METHOD FB_init : BOOL
VAR_INPUT
	bInitRetains : BOOL; // if TRUE, the retain variables are initialized (warm start / cold start)
	bInCopyCode : BOOL;  // if TRUE, the instance afterwards gets moved into the copy code (online change)
END_VAR
nHighestPumpNr := nHighestPumpNr + 1;
nPumpNr := nHighestPumpNr;
END_METHOD

ACTION A_PumpConst:
//Egal in welchem State, wenn Flow neu gesetzt wird, dann Rotate neu senden
//Wenn bStop, in jedem State zu Stop gehen

IF nStateA_Pump = 0 THEN
	nPumpSpeed := nPumpSpeedNew;
	nStateA_Pump := 1;
END_IF

CASE nStateA_Pump OF
	1:	//Motor rechts drehen
		fbTMCM6110(bExecute:= TRUE, eCommand:= E_TMCMCommand.ROTATE_R, nSendValue:= nPumpSpeed, nMotorNr:= nPumpNr);
		IF NOT fbTMCM6110.bBusy THEN
			IF fbTMCM6110.bError THEN
				nStateA_Pump := 99;	
			ELSE
				IF nPumpSpeed = nPumpSpeedNew THEN
					nStateA_Pump := 2;
				ELSE
					nStateA_Pump := 0;
				END_IF
			END_IF
			fbTMCM6110(bExecute:= FALSE, nMotorNr:= nPumpNr);
		END_IF
		
	2:	//IstSpeed abfragen
		fbTMCM6110(bExecute:= TRUE, eCommand:= E_TMCMCommand.GET_ACT_SPEED, nMotorNr:= nPumpNr);
		IF NOT fbTMCM6110.bBusy THEN
			IF fbTMCM6110.bError THEN
				nStateA_Pump := 99;	
			ELSE
				IF nPumpSpeed <> nPumpSpeedNew THEN
					nStateA_Pump := 0;
				ELSE
					IF fbTMCM6110.nReceiveValue = nPumpSpeed THEN	//SollSpeed erreicht
						IF nPumpSpeed = 0 THEN
							nStateA_Pump := 80;
						END_IF
					END_IF
				END_IF
			END_IF
			fbTMCM6110(bExecute:= FALSE, nMotorNr:= nPumpNr);
		END_IF
END_CASE
END_ACTION

METHOD M_Stop : ERRORID
VAR_INPUT
END_VAR
IF bBusy THEN
	bStop := TRUE;
	nPumpSpeedNew := 0;
END_IF
END_METHOD

ACTION A_PumpQuantity:
//Wenn bStop, in jedem State zu Stop gehen
//Vor Absenden des Move-Befehls, Speed setzen
CASE nStateA_Pump OF
	
	0:	//Set Speed
		nPumpSpeed := nPumpSpeedNew;
		fbTMCM6110(bExecute:= TRUE, eCommand:= E_TMCMCommand.SET_SPEED, nSendValue:= nPumpSpeed, nMotorNr:= nPumpNr);
		IF NOT fbTMCM6110.bBusy THEN
			IF fbTMCM6110.bError THEN
				nStateA_Pump := 99;	
			ELSE
				IF bStop THEN
					nStateA_Pump := 80;
				ELSE
					nStateA_Pump := 1;
				END_IF
			END_IF
			fbTMCM6110(bExecute:= FALSE, nMotorNr:= nPumpNr);
		END_IF
		
	1:	//MoveRel
		fbTMCM6110(bExecute:= TRUE, eCommand:= E_TMCMCommand.MOVE_REL, nSendValue:= nPumpMicroSteps, nMotorNr:= nPumpNr);
		IF NOT fbTMCM6110.bBusy THEN
			IF fbTMCM6110.bError THEN
				nStateA_Pump := 99;	
			ELSE
				IF bStop THEN
					nStateA_Pump := 3;
				ELSE
					nStateA_Pump := 2;
				END_IF
			END_IF
			fbTMCM6110(bExecute:= FALSE, nMotorNr:= nPumpNr);
		END_IF
		
	2:	//Warten, bis Position erreicht
		fbTMCM6110(bExecute:= TRUE, eCommand:= E_TMCMCommand.GET_POS_REACHED, nSendValue:= 0, nMotorNr:= nPumpNr);
		IF NOT fbTMCM6110.bBusy THEN
			IF fbTMCM6110.bError THEN
				nStateA_Pump := 99;	
			ELSE
				IF bStop THEN
					nStateA_Pump := 3;	//Stoppen
				ELSE
					IF fbTMCM6110.nReceiveValue = 1 THEN
						nStateA_Pump := 80;	
					END_IF
				END_IF
			END_IF
			fbTMCM6110(bExecute:= FALSE, nMotorNr:= nPumpNr);
		END_IF
		
	3:	//Stoppen
		fbTMCM6110(bExecute:= TRUE, eCommand:= E_TMCMCommand.STOP, nSendValue:= 0, nMotorNr:= nPumpNr);
		IF NOT fbTMCM6110.bBusy THEN
			IF fbTMCM6110.bError THEN
				nStateA_Pump := 99;	
			ELSE
				nStateA_Pump := 80;	
			END_IF
			fbTMCM6110(bExecute:= FALSE, nMotorNr:= nPumpNr);
		END_IF
		
END_CASE
END_ACTION

METHOD M_PumpQuantity : ERRORID
VAR_INPUT
	nQuantity 	: DINT;
	nFlow		: DINT;
END_VAR
bPumpQuantity := TRUE;
nPumpMicroSteps := REAL_TO_DINT(DINT_TO_REAL(nQuantity) * cFactorQuantToMicroSteps);
nPumpSpeedNew := REAL_TO_DINT(DINT_TO_REAL(nFlow) * cFactorFlowToSpeed / cDivisorFlowToSpeed);
bBusy := TRUE;
END_METHOD

END_FUNCTION_BLOCK

// ---- Hardware/LiquidReserve/FB_TMCM6110.TcPOU
FUNCTION_BLOCK FB_TMCM6110
VAR_INPUT
	bExecute	: BOOL;
	eCommand	: E_TMCMCommand;
	nSendValue	: DINT;	
END_VAR
VAR_IN_OUT
	nMotorNr : USINT;
END_VAR
VAR_OUTPUT
	bBusy			: BOOL;
	bError			: BOOL;
	nReceiveValue	: DINT;	
END_VAR
VAR
	fbSendCanMessage 		: FB_SendCanMessage(ADR(CANInterfaceCom.stCanInterfaceBuffer));
	nState					: USINT;
	uByteArr4Dint			: U_ByteArr4_DINT;
END_VAR

IF bExecute THEN

	IF nState = 0 THEN
		bBusy := TRUE;
		fbSendCanMessage.aTxData[0] := UINT_TO_USINT(SHR(eCommand,8)); //Command
		fbSendCanMessage.aTxData[1] := UINT_TO_USINT(eCommand AND 16#00FF); //Type
		fbSendCanMessage.aTxData[2] := nMotorNr - 1; // "0" für Motor1
		//SendValue in Union kopieren
		uByteArr4Dint.nDINT := nSendValue;
		//Bytes aus Union in TxData kopieren (MSB in Byte3....LSB in Byte6)
		fbSendCanMessage.aTxData[3] := uByteArr4Dint.aBytes[3];
		fbSendCanMessage.aTxData[4] := uByteArr4Dint.aBytes[2];
		fbSendCanMessage.aTxData[5] := uByteArr4Dint.aBytes[1];
		fbSendCanMessage.aTxData[6] := uByteArr4Dint.aBytes[0];
		fbSendCanMessage.tTimeout := T#100MS;
		fbSendCanMessage.nTxLength := 8;
		nState := 60;
	END_IF
	
	IF nState = 60 THEN
		fbSendCanMessage(nIdentifierTX:= 16#01, nIdentifierRX:= 16#02, bExecute:= TRUE);
		IF NOT fbSendCanMessage.bBusy THEN
			IF NOT fbSendCanMessage.bError THEN
				//Response auswerten
				IF fbSendCanMessage.aRxData[1] = 100 THEN	//OK ohne Fehler
					//Bytes aus RxData in UNION kopieren (Byte3 in MSB....Byte6 in LSB)
					uByteArr4Dint.aBytes[3] := fbSendCanMessage.aRxData[3];
					uByteArr4Dint.aBytes[2] := fbSendCanMessage.aRxData[4];
					uByteArr4Dint.aBytes[1] := fbSendCanMessage.aRxData[5];
					uByteArr4Dint.aBytes[0] := fbSendCanMessage.aRxData[6];
					//nDint aus UNION in nReceiveValue koipieren
					nReceiveValue := uByteArr4Dint.nDINT;
					nState := 80;
				ELSE
					nState := 99;	
				END_IF
			ELSE
				nState := 99;
			END_IF
			fbSendCanMessage(bExecute:= FALSE);
		END_IF		
	END_IF
	
	IF nState = 80 THEN
		bBusy := FALSE;
	ELSIF nState = 99 THEN
		bBusy := FALSE;
		bError := TRUE;
	END_IF
	
ELSE
	bError := FALSE;
	nState := 0;
	nSendValue := 0;
	nReceiveValue := 0;
END_IF

END_FUNCTION_BLOCK

// ---- Hardware/FBox/FB_HwRefMultiPurpIO.TcPOU
FUNCTION_BLOCK FB_HwRefMultiPurpIO EXTENDS FB_CanNodeBase
VAR_INPUT
END_VAR
VAR_OUTPUT
END_VAR
VAR
END_VAR

IF bNodeEnabled THEN
	SUPER^();
END_IF

//Wenn die analogen Eingänge gemappt sind, dann müssen diese enabled werden.
//Hier sind diese allerdings nicht verfügbar. Wie komme ich an den Mapping-Status?
//IF F_GetMappingStatus(

ACTION A_ResetApp:
IF nStateA_ResetApp = 0 THEN
	fbSdoWrite(sADSNetID:= stAdsAdress.sNetId, nPortNr:= stAdsAdress.nPort,
				nIndex := cUpdateRequest.nIndex, nSubIndex := 0, nDataLength := 1, nData:= 1, bExecute:= TRUE);
	IF NOT fbSdoWrite.bBusy THEN
		IF fbSdoWrite.bError THEN
			nErrorId := fbSdoWrite.nAdsErrorId;
			nErrorId2 := fbSdoWrite.nSdoErrorId;
			nStateA_ResetApp := 99;  //Error
		ELSE
			nStateA_ResetApp := 80;
		END_IF
		fbSdoWrite(bExecute:= FALSE);
	END_IF
END_IF
END_ACTION

END_FUNCTION_BLOCK

// ---- Hardware/FBox/FB_PCV.TcPOU
FUNCTION_BLOCK FB_PCV
VAR_INPUT
END_VAR
VAR_OUTPUT
	bError : BOOL;
	nErrorId : ERRORID;
END_VAR
VAR
	bFill		: BOOL;
	tmrTimeout	: TON;
	bSensor		AT %I* : BOOL; 	//Verknüpfung mit Füllstandssensor
	bDigiOut 	AT %Q* : BOOL; 	//Verknüpfung muss mit Pumpe und StopVentil erfolgen
	bPneuValve	AT %Q* : BOOL;	//Verknüpfung mit Pneumatikventil (nur bei SolenoidPip)	
END_VAR

IF bSensor AND bFill THEN
	{IF defined(variable:cLiquidBottleNrPCV)}
	IF NOT aSensSysLiquidBottle[cLiquidBottleNrPCV] THEN //kein Systemwasser vorhanden
		bError := TRUE;
		nErrorId := E_ErrorIdCmd.ERRORID_LiquidBottleEmpty;
	END_IF
	{ELSE}
	IF NOT aSensSysLiquidBottle[1] THEN //kein Systemwasser vorhanden
		bError := TRUE;
		nErrorId := E_ErrorIdCmd.ERRORID_LiquidBottleEmpty;
	END_IF	
	{END_IF}

	IF NOT bError AND bFill THEN
		tmrTimeout(IN:= TRUE, PT:=T#1M);
		bDigiOut := TRUE;
	ELSE
		tmrTimeout(IN:= FALSE);
		bDigiOut := FALSE;	
	END_IF

	bFill := FALSE;
ELSE
	tmrTimeout(IN:= FALSE);
	bDigiOut := FALSE;	
	tmrTimeout(IN:= FALSE);
END_IF

IF tmrTimeout.Q THEN
	bError := TRUE;
	nErrorId := E_ErrorIdCmd.ERRORID_TimeOutFillPCV;
	bDigiOut := FALSE;
END_IF

METHOD M_Fill
VAR_INPUT
END_VAR
bFill := TRUE;
END_METHOD

METHOD M_Reset
VAR_INPUT
END_VAR
bError := FALSE;
END_METHOD

METHOD M_SwitchPneuValve
VAR_INPUT
	bOn : BOOL;
END_VAR
bPneuValve := bOn;
END_METHOD

PROPERTY P_bPneuValve : BOOL
GET
P_bPneuValve := bPneuValve;
END_GET
END_PROPERTY

END_FUNCTION_BLOCK

// ---- Hardware/Safety/FB_Safety.TcPOU
FUNCTION_BLOCK FB_Safety  EXTENDS FB_SafetyBase

VAR_INPUT
END_VAR

VAR_OUTPUT
	bVoltageSafe			: BOOL;
	bToolTempSafe			: BOOL;
END_VAR

VAR
	bEmergencyStop			AT %I* : BOOL;	//Notaus ist gedrückt
	bInterlockIsLocked		AT %I* : BOOL;	//Interlock ist ordnungsgemäß verriegelt
	bBoxContactsClosed		AT %I* : BOOL;	//Sicherheitskontakte der Sicherheitsbox geschlossen
	bDriveIsSafe			AT %I* : BOOL;	//Sicherheitsrelais der Antriebe haben nicht angezogen
	bMesIsSafe				AT %I* : BOOL;	//Sicherheitsrelais in MES-Box hat nicht angezogen
	 
	nTwinSafeGrpState		AT %I* : USINT;
	
	bRequDriveOn			AT %Q* : BOOL;	//Request an TwinSafe Gruppe die Drives freizugeben (Relais einschalten)
	bRequMesOn				AT %Q* : BOOL;	//Request an TwinSafe Gruppe die MES freizugeben (Relais im HV-Generator einschalten)
	bRequUnlock				AT %Q* : BOOL;	//Request an TwinSafe Gruppe die Sicherheitsbox zu entriegeln

	bErrAckTwinSafeGrp		AT %Q* : BOOL;	//Error in TwinSafe Gruppe zurücksetzen
	bRunStopTwinSafeGrp		AT %Q* : BOOL := TRUE;	//TwinSafe Gruppe starten/stoppen
	
	nSubstate				: USINT := 0;
	nActionState			: USINT := 0;
	eRequestState			: E_SafetyState;
	eOldState				: E_SafetyState; //wird nur für Verlassen von EmergencyStopReleased durch Quit benötigt
											 //muss also beim Übergang in EmergencyStopPressed gemerkt werden
	
	bBoxContacsAvailable	: BOOL;
	bQuit					: BOOL;
	timer					: TON;
	i						: UINT;
	stPosition				: ST_3DPoint;
	
	stError					: ST_Error;
	stActionData			: ST_ActionData;
	
	pXYDrive				: POINTER TO FB_XYDriveBase;
	
END_VAR

VAR CONSTANT
	rSafePositionX			: REAL := 400000.0;
	rSafePositionY			: REAL := 200000.0;
	nSafeTemp				: UINT := 500; //50°C
END_VAR

IF bBoxContacsAvailable THEN
	A_RunWithBoxContacts();
ELSE
	A_RunWithoutBoxContacts();
END_IF

ACTION A_Lock:
stError.POUState := nActionState;
IF nActionState = 0 THEN
	bRequDriveOn := TRUE;
	bRequUnlock := FALSE;
	nActionState := 1;
ELSIF nActionState = 1 THEN
	//Warten, bis Safety bzw. Drive Relais ein
	//hier Timeout erforderlich?
	//was könnte dazu führen, dass das Drive Relay nicht anzieht?
	//wenn gerade in dem Moment, in dem gelockt wird, der Schlüssel des Interlocks betätigt wird
	//oder wenn ein Box Kontakt geöffnet wird
	timer(IN:=TRUE, PT:=T#500MS);
	IF timer.Q THEN
		stError.ErrorId := E_ErrorIdCmd.ERRORID_TimeOut;
		nActionState := 99;
		timer(IN:= FALSE);
	END_IF
	
	IF NOT bDriveIsSafe THEN
		timer(IN:= FALSE);
		//Drives wieder einschalten, wenn sie bereits initialisiert sind
		fbXYDriveList.M_SetCurrentToHead();
		REPEAT
			pXYDrive := fbXYDriveList.M_Get();
			IF pXYDrive > 0 THEN
				IF pXYDrive^.P_bHomed THEN
					pXYDrive^.M_PowerOn();
				END_IF
			END_IF
		UNTIL pXYDrive = 0
		END_REPEAT
		nActionState := 80;
	END_IF
END_IF

//Errorhandling
IF nActionState = 99 THEN
	stError.POU := E_POU.POU_FB_Safety;
	stError.POUAction := E_POUACT.POUACT_A_Lock;
	fbErrorList.M_Add(stError);
END_IF
END_ACTION

ACTION A_ResetError:
IF nActionState = 0 THEN
	bErrAckTwinSafeGrp := TRUE;
	timer(IN:= TRUE, PT:=T#500MS);
	nActionState := 1;
ELSIF nActionState = 1 THEN
	timer();
	IF timer.Q THEN
		timer(IN:= FALSE);
		bErrAckTwinSafeGrp := FALSE;
		nActionState := 99;
	ELSIF nTwinSafeGrpState = 5 THEN
		bErrAckTwinSafeGrp := FALSE;
	ELSIF nTwinSafeGrpState = 1 THEN
		timer(IN:= FALSE);
		nActionState := 80;
		bErrAckTwinSafeGrp := FALSE;
	END_IF
END_IF
END_ACTION

ACTION A_RunWithBoxContacts:
CASE eCurrentState OF
	E_SafetyState.Init:
		//Dieser State wird nur am Anfang einmal durchlaufen und falls die TwinSafe Gruppe in Error ist,
		//wird dieser zurückgesetzt
		IF nSubState = 0 THEN
			bRunStopTwinSafeGrp := TRUE;
			IF nTwinSafeGrpState <> 1 THEN
				nSubState := 1;
			ELSE
				nSubState := 80;
			END_IF
		END_IF
		//Error zurücksetzen
		IF nSubState = 1 THEN
			A_ResetError();
			IF nActionState >= 80 THEN
				IF nActionState = 99 THEN
					nSubState := 99;
				ELSE
					nSubState := 80;
				END_IF
				nActionState := 0;
			END_IF
		END_IF
		//weiterschalten
		IF nSubState >= 80 THEN
			IF nSubState = 99 THEN
				eCurrentState := E_SafetyState.Error;
			ELSE
				//folgende States sind von hier aus möglich
				//1: EmergencyStopPressed wenn Notaustaster gedrückt
				//2: Locked wenn Interlock verriegelt (MES ist dabei egal)
				//3: UnlockedBoxCtcOpen wenn Interlock entriegelt und der Betätiger im Interlock oder ein anderer Sicherheitskontakt unterbrochen
				//4: UnlockedBoxCtcClosed wenn Interlock entriegelt und der Betätiger im Interlock und alle anderen Sicherheitskontakte geschlossen
				IF bEmergencyStop THEN
					eCurrentState := E_SafetyState.EmergencyStopPressed;
					eOldState := E_SafetyState.Init;
				ELSIF bInterlockIsLocked  THEN
					eCurrentState := E_SafetyState.Locked;
				ELSIF NOT bInterlockIsLocked AND NOT bBoxContactsClosed THEN
					eCurrentState := E_SafetyState.UnlockedBoxCtcOpen;
				ELSIF NOT bInterlockIsLocked AND bBoxContactsClosed THEN
					eCurrentState := E_SafetyState.UnlockedBoxCtcClosed;
				END_IF
			END_IF
			nSubState := 0;
		END_IF
	
	E_SafetyState.Locked:
		//folgende States sind von hier aus möglich
		//1: Error wenn: BoxContact geöffnet wird 
		//				 Interlock durch Schlüssel geöffnet wird ("bInterlockIsLocked" wechselt zu false)
		//				 SaftyLogic meldet Error
		//				 A_Unlock() mit State 99(Error) endet
		//2: EmergencyStopPressed wenn Notaustaster gedrückt
		//3: UnlockedBoxCtcClosed wenn A_Unlock() State 80(Succes) endet
		//bRequDriveOn := TRUE;
		IF nSubstate = 0 THEN //wartet auf StateRequest und überwacht
			bRequDriveOn := TRUE;
			IF NOT (bInterlockIsLocked AND bBoxContactsClosed AND nTwinSafeGrpState = 1) THEN //führt zu Error
				eCurrentState := E_SafetyState.Error;
			ELSIF bEmergencyStop THEN
				eCurrentState := E_SafetyState.EmergencyStopPressed;
				eOldState := E_SafetyState.Locked;
			ELSIF eRequestState = E_SafetyState.Unlocked THEN
				nSubstate := 1;
			END_IF
		ELSIF nSubstate = 1 THEN //führt A_Unlock() aus
			A_Unlock();
			IF nActionState >= 80 THEN
				IF nActionState = 99 THEN
					eCurrentState := E_SafetyState.Error;
				ELSE
					eCurrentState := E_SafetyState.UnlockedBoxCtcClosed;
				END_IF
				nSubState := 0;
				nActionState := 0;
			END_IF
		END_IF

		//Wenn dieser State verlassen wird, dann in jedem Fall bRequDriveOn und bRequMesOn zurücknehmen
		IF eCurrentState <> E_SafetyState.Locked THEN
			bRequDriveOn := FALSE;
			bRequMesOn := FALSE;
		END_IF
		
	E_SafetyState.UnlockedBoxCtcClosed:
		//folgende States sind von hier aus möglich
		//1: Error wenn: SaftyLogic meldet Error oder A_Lock() mit State 99 (Error) endet
		//2: EmergencyStopPressed wenn Notaustaster gedrückt
		//3: UnlockedBoxCtcOpen wenn: BoxContact geöffnet wird 
		//							  Interlock durch Schlüssel geöffnet wird ("bInterlockIsLocked" wechselt zu false)
		//4: Locked wenn A_Lock() State 80(Succes) endet

		IF nSubstate = 0 THEN //wartet auf StateRequest und überwacht
			IF nTwinSafeGrpState <> 1 THEN //führt zu Error
				eCurrentState := E_SafetyState.Error;
			ELSIF NOT bBoxContactsClosed THEN
				eCurrentState := E_SafetyState.UnlockedBoxCtcOpen;
				eOldState := E_SafetyState.UnlockedBoxCtcClosed;
			ELSIF bEmergencyStop THEN
				eCurrentState := E_SafetyState.EmergencyStopPressed;
				eOldState := E_SafetyState.UnlockedBoxCtcClosed;
			ELSIF eRequestState = E_SafetyState.Locked THEN
				nSubstate := 1;
			END_IF
		ELSIF nSubstate = 1 THEN //führt A_Lock() aus
			A_Lock();
			IF nActionState >= 80 THEN
				IF nActionState = 99 THEN
					eCurrentState := E_SafetyState.Error;
				ELSE
					eCurrentState := E_SafetyState.Locked;
				END_IF
				nSubState := 0;
				nActionState := 0;
			END_IF
		END_IF
		
	E_SafetyState.UnlockedBoxCtcOpen:
		//folgende States sind von hier aus möglich
		//1: Error wenn: SaftyLogic meldet Error
		//2: EmergencyStopPressed wenn Notaustaster gedrückt wird
		//3: UnlockedBoxCtcClosed wenn BoxContact geschlossen wird
		IF nTwinSafeGrpState <> 1 THEN
			eCurrentState := E_SafetyState.Error;
		ELSIF bEmergencyStop THEN
			eCurrentState := E_SafetyState.EmergencyStopPressed;
			eOldState := E_SafetyState.UnlockedBoxCtcOpen;
		ELSIF bBoxContactsClosed THEN
			eCurrentState := E_SafetyState.UnlockedBoxCtcClosed;
		END_IF
	
	E_SafetyState.EmergencyStopPressed:
		//folgende States sind von hier aus möglich
		//1: Error wenn: SaftyLogic meldet Error
		//2: EmergencyStopReleased wenn der Notaustaster wieder freigegeben wird
		IF nTwinSafeGrpState <> 1 THEN
			stError.POU := E_POU.POU_FB_Safety;
			stError.POUAction := E_POUACT.POUACT_A_RunWithoutBoxContacts;
			stError.ErrorId := E_ErrorIdCmd.ERRORID_TwinSafeGroupError;
			fbErrorList.M_Add(stError);
			eCurrentState := E_SafetyState.Error;
		ELSIF NOT bEmergencyStop THEN
			eCurrentState := E_SafetyState.EmergencyStopReleased;
		END_IF
	E_SafetyState.EmergencyStopReleased:
		//folgende States sind von hier aus möglich
		//1: Error wenn: SaftyLogic meldet Error
		//2: in vorherigen State wechseln wenn Quit
		IF nTwinSafeGrpState <> 1 THEN
			eCurrentState := E_SafetyState.Error;
		ELSIF bQuit THEN
			bQuit := FALSE;
			eCurrentState := eOldState;
		ELSIF bEmergencyStop THEN
			eCurrentState := E_SafetyState.EmergencyStopPressed;
		END_IF
	E_SafetyState.Error:
		IF bQuit THEN
			bQuit := FALSE;
			eCurrentState := E_SafetyState.Init;
		END_IF
END_CASE
END_ACTION

ACTION A_RunWithoutBoxContacts:
//Statemachine Überwachung Interlock und Notauskreis ohne Boxkontakte
//hier gibt es die States "UnlockedBoxCtcOpen" und "UnlockedBoxCtcClosed" nicht, stattdessen gibt es "Unlocked"
CASE eCurrentState OF
	E_SafetyState.Init:
		//Dieser State wird nur am Anfang einmal durchlaufen und falls die TwinSafe Gruppe in Error ist,
		//wird dieser zurückgesetzt
		IF nSubState = 0 THEN
			IF nTwinSafeGrpState <> 1 THEN
				nSubState := 1;
			ELSE
				nSubState := 80;
			END_IF
		END_IF
		//Error zurücksetzen
		IF nSubState = 1 THEN
			A_ResetError();//Fehlermeldung erfolgt in A_ResetError, aber was ist mit Fehlern, die in der TwinSafeGruppe auftreten?
			IF nActionState >= 80 THEN
				IF nActionState = 99 THEN
					nSubState := 99;
				ELSE
					nSubState := 80;
				END_IF
				nActionState := 0;
			END_IF
		END_IF
		//weiterschalten
		IF nSubState >= 80 THEN
			IF nSubState = 99 THEN
				eCurrentState := E_SafetyState.Error;
			ELSE
				//folgende States sind von hier aus möglich
				//1: EmergencyStopPressed wenn Notaustaster gedrückt
				//2: Locked wenn Interlock verriegelt
				//3: Unlocked wenn Interlock entriegelt
				IF bEmergencyStop THEN
					eCurrentState := E_SafetyState.EmergencyStopPressed;
					eOldState := E_SafetyState.Init;
				ELSIF bInterlockIsLocked  THEN
					eCurrentState := E_SafetyState.Locked;
				ELSIF NOT bInterlockIsLocked  THEN
					eCurrentState := E_SafetyState.Unlocked;
				END_IF
			END_IF
			nSubState := 0;
		END_IF
	
	E_SafetyState.Locked:
		//folgende States sind von hier aus möglich
		//1: Error wenn: Interlock durch Schlüssel geöffnet wird ("bInterlockIsLocked" wechselt zu false)
		//				 SaftyLogic meldet Error
		//				 A_Unlock() mit State 99(Error) endet
		//2: EmergencyStopPressed wenn Notaustaster gedrückt
		//3: Unlocked wenn A_Unlock() State 80(Succes) endet
		IF nSubstate = 0 THEN //wartet auf StateRequest und überwacht
			bRequDriveOn := TRUE;
			IF NOT (bInterlockIsLocked AND nTwinSafeGrpState = 1) THEN //führt zu Error
				//Schlüssel des Interlocks wurde betätigt oder Drahtbruch
				stError.POU := E_POU.POU_FB_Safety;
				stError.POUAction := E_POUACT.POUACT_A_RunWithoutBoxContacts;
				stError.ErrorId := E_ErrorIdCmd.ERRORID_InterlockError;
				fbErrorList.M_Add(stError); 
				eCurrentState := E_SafetyState.Error;
			ELSIF nTwinSafeGrpState <> 1 THEN
				//TwinSafeGruppe ist in Error gegangen
				stError.POU := E_POU.POU_FB_Safety;
				stError.POUAction := E_POUACT.POUACT_A_RunWithoutBoxContacts;
				stError.ErrorId := E_ErrorIdCmd.ERRORID_TwinSafeGroupError;
				fbErrorList.M_Add(stError);
				eCurrentState := E_SafetyState.Error;
			ELSIF bEmergencyStop THEN
				eCurrentState := E_SafetyState.EmergencyStopPressed;
				eOldState := E_SafetyState.Locked;
			ELSIF eRequestState = E_SafetyState.Unlocked THEN
				nSubstate := 1;
			END_IF
		ELSIF nSubstate = 1 THEN //führt A_Unlock() aus
			A_Unlock();
			IF nActionState >= 80 THEN
				IF nActionState = 99 THEN
					//Fehlermeldung erfolgt in A_Unlock
					eCurrentState := E_SafetyState.Error;
				ELSE
					eCurrentState := E_SafetyState.Unlocked;
				END_IF
				nSubState := 0;
				nActionState := 0;
			END_IF
		END_IF

		//Wenn dieser State verlassen wird, dann in jedem Fall bRequDriveOn und bRequMesOn zurücknehmen
		IF eCurrentState <> E_SafetyState.Locked THEN
			bRequDriveOn := FALSE;
			bRequMesOn := FALSE;
		END_IF
		
	E_SafetyState.Unlocked:
		//folgende States sind von hier aus möglich
		//1: Error wenn: SafetyLogic meldet Error oder A_Locked() mit State 99 (Error) endet
		//2: EmergencyStopPressed wenn Notaustaster gedrückt
		//3: Locked wenn A_Lock() State 80(Succes) endet

		IF nSubstate = 0 THEN //wartet auf StateRequest und überwacht
			//wieso soll bInterlockIsLocked zu Error führen?
			//kann  bInterlockIsLocked in diesem State eigentlich gesetzt werden?
			//Drahtbruch führt nicht zu Gruppenfehler, da Stommessung und Testpulse aus
			IF bInterlockIsLocked THEN
				stError.POU := E_POU.POU_FB_Safety;
				stError.POUAction := E_POUACT.POUACT_A_RunWithoutBoxContacts;
				stError.ErrorId := E_ErrorIdCmd.ERRORID_InterlockError;
				fbErrorList.M_Add(stError);
				eCurrentState := E_SafetyState.Error;
			ELSIF nTwinSafeGrpState <> 1 THEN //führt zu Error
				stError.POU := E_POU.POU_FB_Safety;
				stError.POUAction := E_POUACT.POUACT_A_RunWithoutBoxContacts;
				stError.ErrorId := E_ErrorIdCmd.ERRORID_TwinSafeGroupError;
				fbErrorList.M_Add(stError);
				eCurrentState := E_SafetyState.Error;
			ELSIF bEmergencyStop THEN
				eCurrentState := E_SafetyState.EmergencyStopPressed;
				eOldState := E_SafetyState.Unlocked;
			ELSIF eRequestState = E_SafetyState.Locked THEN
				nSubstate := 1;
			END_IF
		ELSIF nSubstate = 1 THEN //führt A_Lock() aus
			A_Lock();
			IF nActionState >= 80 THEN
				IF nActionState = 99 THEN
					//Fehlermeldung erfolgt in A_Lock
					eCurrentState := E_SafetyState.Error;
				ELSE
					eCurrentState := E_SafetyState.Locked;
				END_IF
				nSubState := 0;
				nActionState := 0;
			END_IF
		END_IF
	
	E_SafetyState.EmergencyStopPressed:
		//folgende States sind von hier aus möglich
		//1: Error wenn: SaftyLogic meldet Error
		//2: EmergencyStopReleased wenn der Notaustaster wieder freigegeben wird
		IF nTwinSafeGrpState <> 1 THEN
			stError.POU := E_POU.POU_FB_Safety;
			stError.POUAction := E_POUACT.POUACT_A_RunWithoutBoxContacts;
			stError.ErrorId := E_ErrorIdCmd.ERRORID_TwinSafeGroupError;
			fbErrorList.M_Add(stError);
			eCurrentState := E_SafetyState.Error;
		ELSIF NOT bEmergencyStop THEN
			eCurrentState := E_SafetyState.EmergencyStopReleased;
		END_IF
	E_SafetyState.EmergencyStopReleased:
		//folgende States sind von hier aus möglich
		//1: Error wenn: SaftyLogic meldet Error
		//2: in vorherigen State wechseln wenn Quit
		IF nTwinSafeGrpState <> 1 THEN
			eCurrentState := E_SafetyState.Error;
		ELSIF bQuit THEN
			bQuit := FALSE;
			eCurrentState := eOldState;
		ELSIF bEmergencyStop THEN
			eCurrentState := E_SafetyState.EmergencyStopPressed;
		END_IF
	E_SafetyState.Error:
		IF bQuit THEN
			bQuit := FALSE;
			eCurrentState := E_SafetyState.Init;
		END_IF
END_CASE
END_ACTION

ACTION A_Unlock:
//1. Hochspannung ausschalten
//2. Fall Tools temperiert, in sichere Position fahren
//3. warten bis o.g. Bedingungen erfüllt (Timeout)
//4. Antriebe ausschalten
//5. Interlock entriegeln
stError.POUState := nActionState;
CASE nActionState OF
	0:	//GCode aktiv?
		IF GCode.bBusy THEN
			GCode.M_Stop();
		ELSE
			nActionState := 1;
		END_IF
		
	1:	//Hochspannung aus
		{IF defined(variable:fbHighVoltSupplyRef)}
		 fbHighVoltSupplyRef.M_SwitchVoltage(1,FALSE);
		 fbHighVoltSupplyRef.M_SwitchVoltage(2,FALSE);
		{END_IF}
		bRequMesOn := FALSE; //Relais in HV-Generator abschalten
		nActionState := 3;
		//Tools temperiert?
		FOR i:= 1 TO fbObjectDirectory.nCntMZHead BY 1 DO
			IF afbMzHead[i].P_bIsHot THEN
				nActionState := 2;
				stActionData.eAction := E_Action.ACTION_MoveAllHome;
				stError.ErrorId := fbComplexAction.M_ExeAction(stActionData);
				IF stError.ErrorId > 0 THEN
					nActionState := 99;
					EXIT;
				END_IF
			END_IF
		END_FOR
		
	2:	//MoveAllHome ready?
		IF NOT fbComplexAction.bBusy THEN
			IF fbComplexAction.bError THEN
				stError.ErrorId := fbComplexAction.nErrorId; 
			ELSE
				nActionState := 3;
			END_IF
		END_IF
 		
	3:	//Spannungsfreiheit Hochspannungsmodul?
		nActionState := 4;
		{IF defined(variable:fbHighVoltSupplyRef)}
		//>20 um Rauschen des analogen Eingangs zu unterbinden
		IF fbHighVoltSupplyRef.bHVPSAvailable AND NOT fbHighVoltSupplyRef.bSafeVoltage AND (fbHighVoltSupplyRef.M_GetVoltage() > 20) THEN
			nActionState := 3;
		END_IF
		{END_IF}
		
	4:	//Antriebe ausschalten
		fbXYDriveList.M_SetCurrentToHead();
		REPEAT
			pXYDrive := fbXYDriveList.M_Get();
			IF pXYDrive > 0 THEN
				pXYDrive^.M_PowerOff();
			END_IF
		UNTIL pXYDrive = 0
		END_REPEAT	
		nActionState := 5;
		
	5:	//Safety bzw. Drive Relais ausschalten und Interlock entriegeln
		bRequDriveOn := FALSE;
		bRequUnlock := TRUE;
		nActionState := 6;
		
	6:	//Warten bis Interlock entriegelt
		timer(IN:=TRUE, PT:=T#500MS);
		IF timer.Q THEN
			stError.ErrorId := E_ErrorIdCmd.ERRORID_TimeOut;
			nActionState := 99;
			timer(IN:= FALSE);
		END_IF
		
		IF NOT bInterlockIsLocked THEN
			timer(IN:= FALSE);
			nActionState := 80;
		END_IF	
END_CASE

//Errorhandling
IF nActionState = 99 THEN
	stError.POU := E_POU.POU_FB_Safety;
	stError.POUAction := E_POUACT.POUACT_A_Unlock;
	fbErrorList.M_Add(stError);
END_IF
END_ACTION

METHOD M_CheckBoxCtcMapping
VAR_INPUT
END_VAR
IF F_GetMappingStatus(ADR(bBoxContactsClosed),SIZEOF(bBoxContactsClosed)) = EPlcMappingStatus.MS_Partial THEN
	bBoxContacsAvailable := TRUE;
END_IF
END_METHOD

METHOD M_Control : ERRORID
VAR_INPUT
	eCtrl : E_SafetyCtrl;
END_VAR
CASE eCurrentState OF
	E_SafetyState.Init:
		//kein Befehl erlaubt, Meldung InvalidState
	E_SafetyState.Locked:
		//erlaubt ist Unlock
		IF eCtrl = E_SafetyCtrl.Unlock THEN
			eRequestState := E_SafetyState.Unlocked;
		ELSE
			M_Control := E_ErrorIdCmd.ERRORID_InvalidSafetyState;
		END_IF
	E_SafetyState.UnlockedBoxCtcClosed,E_SafetyState.Unlocked:
		//erlaubt ist Lock
		IF eCtrl = E_SafetyCtrl.Lock THEN
			eRequestState := E_SafetyState.Locked;
		ELSE
			M_Control := E_ErrorIdCmd.ERRORID_InvalidSafetyState;
		END_IF
	E_SafetyState.UnlockedBoxCtcOpen:
		M_Control := E_ErrorIdCmd.ERRORID_InvalidSafetyState;
	E_SafetyState.EmergencyStopPressed:
		M_Control := E_ErrorIdCmd.ERRORID_InvalidSafetyState;
	E_SafetyState.EmergencyStopReleased,E_SafetyState.Error:
		//erlaubt ist nur Quit
		IF eCtrl = E_SafetyCtrl.Quit THEN
			bQuit := TRUE;
		ELSE
			M_Control := E_ErrorIdCmd.ERRORID_InvalidSafetyState;
		END_IF
END_CASE
END_METHOD

METHOD M_MesBoxOn : ERRORID
VAR_INPUT
END_VAR
IF eCurrentState = E_SafetyState.Locked THEN
	bRequMesOn := TRUE;
ELSE
	M_MesBoxOn := E_ErrorIdCmd.ERRORID_InvalidSafetyState;
END_IF
END_METHOD

PROPERTY P_nSafeToolTemp : UINT
GET
P_nSafeToolTemp := nSafeTemp;
END_GET
END_PROPERTY

PROPERTY P_rSafePositionX : REAL
GET
P_rSafePositionX := rSafePositionX;
END_GET
END_PROPERTY

PROPERTY P_rSafePositionY : REAL
GET
P_rSafePositionY := rSafePositionY;
END_GET
END_PROPERTY

END_FUNCTION_BLOCK

// ---- Hardware/Safety/FB_SafetyBase.TcPOU
FUNCTION_BLOCK FB_SafetyBase
VAR_INPUT
END_VAR
VAR_OUTPUT
	eCurrentState : E_SafetyState;
END_VAR
VAR
END_VAR

eCurrentState := E_SafetyState.Locked;

METHOD M_Control : ERRORID
VAR_INPUT
	eCtrl : E_SafetyCtrl;
END_VAR
END_METHOD

METHOD M_MesBoxOn : ERRORID
VAR_INPUT
END_VAR
END_METHOD

END_FUNCTION_BLOCK

// ---- Hardware/Safety/FB_SafetyPseudo.TcPOU
FUNCTION_BLOCK FB_SafetyPseudo EXTENDS FB_SafetyBase
VAR
	bInput 	AT %I* : BOOL;
	bOutput AT %Q* : BOOL;
	nState : USINT;
	pXYDrive : POINTER TO FB_XYDriveBase;
END_VAR
VAR_OUTPUT
	
END_VAR

//Überwachung der Verriegelung ohne TwinSafe (derzeit nur in RPD IWS in Benutzung)
//Wenn Verriegelung durch Schlüssel oder mit Gewalt geöffnet wird, dann müssen die Antriebe
//gestoppt werden -> QuickStop -> PowerOFF
//QuickStop nur wenn Motion aktiv

CASE nState OF
	0:	//Überwachung im verriegelten Zustand
		IF NOT bInput THEN
			eCurrentState := E_SafetyState.Unlocked;
			fbXYDriveList.M_SetCurrentToHead();
			REPEAT
				pXYDrive := fbXYDriveList.M_Get();
				IF pXYDrive > 0 THEN
					pXYDrive^.M_Stop();
				END_IF
			UNTIL pXYDrive = 0
			END_REPEAT			
			nState := 1;
		END_IF
	1:
		fbXYDriveList.M_SetCurrentToHead();
		REPEAT
			pXYDrive := fbXYDriveList.M_Get();
			IF pXYDrive > 0 THEN
				pXYDrive^.M_PowerOff();
			END_IF
		UNTIL pXYDrive = 0
		END_REPEAT			
	
	10:	//Verriegeln
		//Unter welchen Bedingungen darf verrieglt werden?
		IF bInput THEN
			eCurrentState := E_SafetyState.Locked;
			nState := 0;
			fbXYDriveList.M_SetCurrentToHead();
			REPEAT
				pXYDrive := fbXYDriveList.M_Get();
				IF pXYDrive > 0 THEN
					IF pXYDrive^.P_bHomed AND NOT pXYDrive^.P_bError THEN
						pXYDrive^.M_PowerOn();
					END_IF
 				END_IF
			UNTIL pXYDrive = 0
			END_REPEAT			
		END_IF
	
	20: //Entriegelt
END_CASE

METHOD FB_init : BOOL
VAR_INPUT
	bInitRetains : BOOL; // if TRUE, the retain variables are initialized (warm start / cold start)
	bInCopyCode : BOOL;  // if TRUE, the instance afterwards gets moved into the copy code (online change)
END_VAR
eCurrentState := E_SafetyState.Locked;
END_METHOD

END_FUNCTION_BLOCK

// ---- Hardware/Safety/FB_SafetyStacker.TcPOU
FUNCTION_BLOCK FB_SafetyStacker  EXTENDS FB_SafetyBase

VAR_INPUT
END_VAR

VAR_OUTPUT
	bVoltageSafe			: BOOL;
	bToolTempSafe			: BOOL;
END_VAR

VAR
	bEmergencyStop			AT %I* : BOOL;	//Notaus ist gedrückt
	bInterlockIsLocked		AT %I* : BOOL;	//Interlock ist ordnungsgemäß verriegelt
	bBoxContactsClosed		AT %I* : BOOL;	//Sicherheitskontakte der Sicherheitsbox geschlossen
	bDriveIsSafe			AT %I* : BOOL;	//Sicherheitsrelais für Antriebe nicht angezogen
	 
	nTwinSafeGrpState		AT %I* : USINT;
	
	bRequDriveOn			AT %Q* : BOOL;	//Request an TwinSafe Gruppe die Drives freizugeben (Relais einschalten)
	bRequUnlock				AT %Q* : BOOL;	//Request an TwinSafe Gruppe die Sicherheitsbox zu entriegeln

	bErrAckTwinSafeGrp		AT %Q* : BOOL;	//Error in TwinSafe Gruppe zurücksetzen
	bRunStopTwinSafeGrp		AT %Q* : BOOL := TRUE;	//TwinSafe Gruppe starten/stoppen
	
	nSubstate				: USINT := 0;
	nActionState			: USINT := 0;
	eRequestState			: E_SafetyState;
	eOldState				: E_SafetyState; //wird nur für Verlassen von EmergencyStopReleased durch Quit benötigt
											 //muss also beim Übergang in EmergencyStopPressed gemerkt werden
	
	bQuit					: BOOL;
	timer					: TON;
	i						: UINT;
	
	stError					: ST_Error;
	stActionData			: ST_ActionData;
	
	pHwRef_SpinDrive		: POINTER TO FB_HwRefEL70xxDrive;
	pHwRef_LiftDrive		: POINTER TO FB_HwRefEL70xxDrive;

	fbEL70xxPower			: FB_HWECtrl_EL70xx_Power;
	fbEL70xxHoming			: FB_HWECtrl_EL70xx_Home; //nur für SpinDrive
	bSpinDriveWasInit		: BOOL;
	bLiftDriveWasInit		: BOOL;
	
END_VAR

CASE eCurrentState OF
	E_SafetyState.Init:
		//Dieser State wird nur am Anfang einmal durchlaufen und falls die TwinSafe Gruppe in Error ist,
		//wird dieser zurückgesetzt
		IF nSubState = 0 THEN
			bRunStopTwinSafeGrp := TRUE;
			IF nTwinSafeGrpState <> 1 THEN
				nSubState := 1;
			ELSE
				nSubState := 80;
			END_IF
		END_IF
		//Error zurücksetzen
		IF nSubState = 1 THEN
			A_ResetError();
			IF nActionState >= 80 THEN
				IF nActionState = 99 THEN
					nSubState := 99;
				ELSE
					nSubState := 80;
				END_IF
				nActionState := 0;
			END_IF
		END_IF
		//weiterschalten
		IF nSubState >= 80 THEN
			IF nSubState = 99 THEN
				eCurrentState := E_SafetyState.Error;
			ELSE
				//folgende States sind von hier aus möglich
				//1: EmergencyStopPressed wenn Notaustaster gedrückt
				//2: Locked wenn Interlock verriegelt
				//3: UnlockedBoxCtcOpen wenn Interlock entriegelt und der Betätiger im Interlock oder ein anderer Sicherheitskontakt unterbrochen
				//4: UnlockedBoxCtcClosed wenn Interlock entriegelt und der Betätiger im Interlock und alle anderen Sicherheitskontakte geschlossen
				IF bEmergencyStop THEN
					eCurrentState := E_SafetyState.EmergencyStopPressed;
					eOldState := E_SafetyState.Init;
				ELSIF bInterlockIsLocked  THEN
					eCurrentState := E_SafetyState.Locked;
				ELSIF NOT bInterlockIsLocked AND NOT bBoxContactsClosed THEN
					eCurrentState := E_SafetyState.UnlockedBoxCtcOpen;
				ELSIF NOT bInterlockIsLocked AND bBoxContactsClosed THEN
					eCurrentState := E_SafetyState.UnlockedBoxCtcClosed;
				END_IF
			END_IF
			nSubState := 0;
		END_IF
	
	E_SafetyState.Locked:
		//folgende States sind von hier aus möglich
		//1: Error wenn: BoxContact geöffnet wird 
		//				 Interlock durch Schlüssel geöffnet wird ("bInterlockIsLocked" wechselt zu false)
		//				 SaftyLogic meldet Error
		//				 A_Unlock() mit State 99(Error) endet
		//2: EmergencyStopPressed wenn Notaustaster gedrückt
		//3: UnlockedBoxCtcClosed wenn A_Unlock() State 80(Succes) endet
		//bRequDriveOn := TRUE;
		IF nSubstate = 0 THEN //wartet auf StateRequest und überwacht
			bRequDriveOn := TRUE;
			IF NOT (bInterlockIsLocked AND bBoxContactsClosed AND nTwinSafeGrpState = 1) THEN //führt zu Error
				eCurrentState := E_SafetyState.Error;
			ELSIF bEmergencyStop THEN
				eCurrentState := E_SafetyState.EmergencyStopPressed;
				eOldState := E_SafetyState.Locked;
			ELSIF eRequestState = E_SafetyState.Unlocked THEN
				nSubstate := 1;
			END_IF
		ELSIF nSubstate = 1 THEN //führt A_Unlock() aus
			A_Unlock();
			IF nActionState >= 80 THEN
				IF nActionState = 99 THEN
					eCurrentState := E_SafetyState.Error;
				ELSE
					eCurrentState := E_SafetyState.UnlockedBoxCtcClosed;
				END_IF
				nSubState := 0;
				nActionState := 0;
			END_IF
		END_IF

		//Wenn dieser State verlassen wird, dann in jedem Fall bRequDriveOn und bRequMesOn zurücknehmen
		IF eCurrentState <> E_SafetyState.Locked THEN
			bRequDriveOn := FALSE;
		END_IF
		
	E_SafetyState.UnlockedBoxCtcClosed:
		//folgende States sind von hier aus möglich
		//1: Error wenn: SaftyLogic meldet Error oder A_Lock() mit State 99 (Error) endet
		//2: EmergencyStopPressed wenn Notaustaster gedrückt
		//3: UnlockedBoxCtcOpen wenn: BoxContact geöffnet wird 
		//							  Interlock durch Schlüssel geöffnet wird ("bInterlockIsLocked" wechselt zu false)
		//4: Locked wenn A_Lock() State 80(Succes) endet

		IF nSubstate = 0 THEN //wartet auf StateRequest und überwacht
			IF nTwinSafeGrpState <> 1 THEN //führt zu Error
				eCurrentState := E_SafetyState.Error;
			ELSIF NOT bBoxContactsClosed THEN
				eCurrentState := E_SafetyState.UnlockedBoxCtcOpen;
				eOldState := E_SafetyState.UnlockedBoxCtcClosed;
			ELSIF bEmergencyStop THEN
				eCurrentState := E_SafetyState.EmergencyStopPressed;
				eOldState := E_SafetyState.UnlockedBoxCtcClosed;
			ELSIF eRequestState = E_SafetyState.Locked THEN
				nSubstate := 1;
			END_IF
		ELSIF nSubstate = 1 THEN //führt A_Lock() aus
			A_Lock();
			IF nActionState >= 80 THEN
				IF nActionState = 99 THEN
					eCurrentState := E_SafetyState.Error;
				ELSE
					eCurrentState := E_SafetyState.Locked;
				END_IF
				nSubState := 0;
				nActionState := 0;
			END_IF
		END_IF
		
	E_SafetyState.UnlockedBoxCtcOpen:
		//folgende States sind von hier aus möglich
		//1: Error wenn: SaftyLogic meldet Error
		//2: EmergencyStopPressed wenn Notaustaster gedrückt wird
		//3: UnlockedBoxCtcClosed wenn BoxContact geschlossen wird
		IF nTwinSafeGrpState <> 1 THEN
			eCurrentState := E_SafetyState.Error;
		ELSIF bEmergencyStop THEN
			eCurrentState := E_SafetyState.EmergencyStopPressed;
			eOldState := E_SafetyState.UnlockedBoxCtcOpen;
		ELSIF bBoxContactsClosed THEN
			eCurrentState := E_SafetyState.UnlockedBoxCtcClosed;
		END_IF
	
	E_SafetyState.EmergencyStopPressed:
		//folgende States sind von hier aus möglich
		//1: Error wenn: SaftyLogic meldet Error
		//2: EmergencyStopReleased wenn der Notaustaster wieder freigegeben wird
		IF nTwinSafeGrpState <> 1 THEN
			stError.POU := E_POU.POU_FB_Safety;
			stError.POUAction := E_POUACT.POUACT_A_RunWithoutBoxContacts;
			stError.ErrorId := E_ErrorIdCmd.ERRORID_TwinSafeGroupError;
			fbErrorList.M_Add(stError);
			eCurrentState := E_SafetyState.Error;
		ELSIF NOT bEmergencyStop THEN
			eCurrentState := E_SafetyState.EmergencyStopReleased;
		END_IF
	E_SafetyState.EmergencyStopReleased:
		//folgende States sind von hier aus möglich
		//1: Error wenn: SaftyLogic meldet Error
		//2: in vorherigen State wechseln wenn Quit
		IF nTwinSafeGrpState <> 1 THEN
			eCurrentState := E_SafetyState.Error;
		ELSIF bQuit THEN
			bQuit := FALSE;
			eCurrentState := eOldState;
		ELSIF bEmergencyStop THEN
			eCurrentState := E_SafetyState.EmergencyStopPressed;
		END_IF
	E_SafetyState.Error:
		IF bQuit THEN
			bQuit := FALSE;
			eCurrentState := E_SafetyState.Init;
		END_IF
END_CASE

ACTION A_Lock:
stError.POUState := nActionState;
IF nActionState = 0 THEN
	bRequDriveOn := TRUE;
	bRequUnlock := FALSE;
	nActionState := 1;
ELSIF nActionState = 1 THEN
	//Warten, bis Safety bzw. Drive Relais ein
	//hier Timeout erforderlich?
	//was könnte dazu führen, dass das Drive Relay nicht anzieht?
	//wenn gerade in dem Moment, in dem gelockt wird, der Schlüssel des Interlocks betätigt wird
	//oder wenn ein Box Kontakt geöffnet wird
	timer(IN:=TRUE, PT:=T#500MS);
	IF timer.Q THEN
		stError.ErrorId := E_ErrorIdCmd.ERRORID_TimeOut;
		nActionState := 99;
		timer(IN:= FALSE);
	END_IF
	
	IF NOT bDriveIsSafe THEN
		timer(IN:= FALSE);
		//Drives wieder einschalten, wenn sie bereits initialisiert waren
		IF bSpinDriveWasInit OR bLiftDriveWasInit THEN
			nActionState := 2;
		ELSE
			nActionState := 80;	
		END_IF
	END_IF
	
ELSIF nActionState = 2 THEN //Power SpinDrive
	{IF defined(variable:fbHwRefSpinDrive)}
	pHwRef_SpinDrive := ADR(fbHwRefSpinDrive);
	fbEL70xxPower(pHwRef:= pHwRef_SpinDrive, bEnable:= TRUE, bExecute:= TRUE);
	IF NOT fbEL70xxPower.bBusy THEN
		fbEL70xxPower(pHwRef:= pHwRef_SpinDrive, bExecute:= FALSE);
		nActionState := 3;
	END_IF
	{ELSE}
		nActionState := 3;
	{END_IF}
ELSIF nActionState = 3 THEN //Power LiftDrive
	{IF defined(variable:fbHwRefLiftDrive)}
	pHwRef_LiftDrive := ADR(fbHwRefLiftDrive);
	fbEL70xxPower(pHwRef:= pHwRef_LiftDrive, bEnable:= TRUE, bExecute:= TRUE);
	IF NOT fbEL70xxPower.bBusy THEN
		fbEL70xxPower(pHwRef:= pHwRef_LiftDrive, bExecute:= FALSE);
		nActionState := 4;
	END_IF	
	{ELSE}
		nActionState := 4;
	{END_IF}
ELSIF nActionState = 4 THEN //Homing SpinDrive
	{IF defined(variable:fbHwRefSpinDrive)}
	fbEL70xxHoming(pHwRef:= pHwRef_SpinDrive, bExecute:= TRUE);
	IF NOT fbEL70xxHoming.bBusy THEN
		IF fbEL70xxHoming.bError THEN
			stError.ErrorId := fbEL70xxHoming.nErrorId;
			nActionState := 99;
		ELSE
			nActionState := 80;
		END_IF
		fbEL70xxHoming(pHwRef:= pHwRef_SpinDrive, bExecute:= FALSE);
	END_IF
	{ELSE}
		nActionState := 80;
	{END_IF}
END_IF

//Errorhandling
IF nActionState = 99 THEN
	stError.POU := E_POU.POU_FB_Safety;
	stError.POUAction := E_POUACT.POUACT_A_Lock;
	fbErrorList.M_Add(stError);
END_IF
END_ACTION

ACTION A_ResetError:
IF nActionState = 0 THEN
	bErrAckTwinSafeGrp := TRUE;
	timer(IN:= TRUE, PT:=T#500MS);
	nActionState := 1;
ELSIF nActionState = 1 THEN
	timer();
	IF timer.Q THEN
		timer(IN:= FALSE);
		bErrAckTwinSafeGrp := FALSE;
		nActionState := 99;
	ELSIF nTwinSafeGrpState = 5 THEN
		bErrAckTwinSafeGrp := FALSE;
	ELSIF nTwinSafeGrpState = 1 THEN
		timer(IN:= FALSE);
		nActionState := 80;
		bErrAckTwinSafeGrp := FALSE;
	END_IF
END_IF
END_ACTION

ACTION A_Unlock:
//1. Antriebe ausschalten (nur Spin- und LiftDrive)
//2. Interlock entriegeln
stError.POUState := nActionState;
CASE nActionState OF
	0:	//Antriebe ausschalten
		//vorher merken, ob Drive initialiert war
		{IF defined(variable:fbHwRefSpinDrive)}
		pHwRef_SpinDrive := ADR(fbHwRefSpinDrive);
		bSpinDriveWasInit := pHwRef_SpinDrive^.P_bIsInit;
		fbEL70xxPower(pHwRef:= pHwRef_SpinDrive, bEnable:= FALSE, bExecute:= TRUE);
		IF NOT fbEL70xxPower.bBusy THEN
			fbEL70xxPower(pHwRef:= pHwRef_SpinDrive, bExecute:= FALSE);
			nActionState := 1;
		END_IF
		{ELSE}
		nActionState := 1;
		{END_IF}
		
	1:	{IF defined(variable:fbHwRefLiftDrive)}
		pHwRef_LiftDrive := ADR(fbHwRefLiftDrive);
		bLiftDriveWasInit := pHwRef_LiftDrive^.P_bIsInit;
		fbEL70xxPower(pHwRef:= pHwRef_LiftDrive, bEnable:= FALSE, bExecute:= TRUE);
		IF NOT fbEL70xxPower.bBusy THEN
			fbEL70xxPower(pHwRef:= pHwRef_LiftDrive, bExecute:= FALSE);
			nActionState := 2;
		END_IF
		{ELSE}
		nActionState := 2;
		{END_IF}
		
	2:	//Safety bzw. Drive Relais ausschalten und Interlock entriegeln
		bRequDriveOn := FALSE;
		bRequUnlock := TRUE;
		nActionState := 3;
		
	3:	//Warten bis Interlock entriegelt
		timer(IN:=TRUE, PT:=T#500MS);
		IF timer.Q THEN
			stError.ErrorId := E_ErrorIdCmd.ERRORID_TimeOut;
			nActionState := 99;
			timer(IN:= FALSE);
		END_IF
		
		IF NOT bInterlockIsLocked THEN
			timer(IN:= FALSE);
			nActionState := 80;
		END_IF	
END_CASE

//Errorhandling
IF nActionState = 99 THEN
	stError.POU := E_POU.POU_FB_Safety;
	stError.POUAction := E_POUACT.POUACT_A_Unlock;
	fbErrorList.M_Add(stError);
END_IF
END_ACTION

METHOD M_Control : ERRORID
VAR_INPUT
	eCtrl : E_SafetyCtrl;
END_VAR
CASE eCurrentState OF
	E_SafetyState.Init:
		//kein Befehl erlaubt, Meldung InvalidState
	E_SafetyState.Locked:
		//die beiden Drives dürfen nicht aktiv sein
		{IF defined(variable:fbHwRefSpinDrive)}
		pHwRef_SpinDrive := ADR(fbHwRefSpinDrive);
		{END_IF}
		
		{IF defined(variable:fbHwRefSpinDrive)}
		pHwRef_LiftDrive := ADR(fbHwRefLiftDrive);
		{END_IF}
		
		IF pHwRef_SpinDrive > 0 AND_THEN pHwRef_SpinDrive^.P_bBusy THEN
			RETURN;
		END_IF
		
		IF pHwRef_LiftDrive > 0 AND_THEN pHwRef_LiftDrive^.P_bBusy THEN
			RETURN;
		END_IF
		
		IF eCtrl = E_SafetyCtrl.Unlock THEN
			eRequestState := E_SafetyState.Unlocked;
		ELSE
			M_Control := E_ErrorIdCmd.ERRORID_InvalidSafetyState;
		END_IF
	E_SafetyState.UnlockedBoxCtcClosed,E_SafetyState.Unlocked:
		//erlaubt ist Lock
		IF eCtrl = E_SafetyCtrl.Lock THEN
			eRequestState := E_SafetyState.Locked;
		ELSE
			M_Control := E_ErrorIdCmd.ERRORID_InvalidSafetyState;
		END_IF
	E_SafetyState.UnlockedBoxCtcOpen:
		M_Control := E_ErrorIdCmd.ERRORID_InvalidSafetyState;
	E_SafetyState.EmergencyStopPressed:
		M_Control := E_ErrorIdCmd.ERRORID_InvalidSafetyState;
	E_SafetyState.EmergencyStopReleased,E_SafetyState.Error:
		//erlaubt ist nur Quit
		IF eCtrl = E_SafetyCtrl.Quit THEN
			bQuit := TRUE;
		ELSE
			M_Control := E_ErrorIdCmd.ERRORID_InvalidSafetyState;
		END_IF
END_CASE
END_METHOD

END_FUNCTION_BLOCK

// ---- Hardware/Safety/FB_SignalLight.TcPOU
FUNCTION_BLOCK FB_SignalLight
VAR_INPUT
	eSafetyState	: E_SafetyState;
	eMachineState 	: E_MachineState;	
END_VAR
VAR_OUTPUT
END_VAR
VAR
	//Blink
	tmrBlink : TON;
	nStateBlink : USINT;
	bBlink	: BOOL;
	
	//Ausgänge für LEDs
	bRed 	AT %Q* : BOOL;
	bYellow AT %Q* : BOOL;
	bGreen	AT %Q* : BOOL;
END_VAR

A_Blink();
IF eSafetyState = E_SafetyState.EmergencyStopPressed THEN
	//rot blinkend
	bRed := TRUE AND bBlink;
	bYellow := FALSE;
	bGreen := FALSE;
	RETURN;
END_IF

CASE eMachineState OF
	E_MachineState.MACHINESTATE_Active, E_MachineState.MACHINESTATE_Running:
		bRed := FALSE;
		bYellow := FALSE;
		bGreen := TRUE;
	E_MachineState.MACHINESTATE_Error:
		bRed := TRUE;
		bYellow := FALSE;
		bGreen := FALSE;		
	E_MachineState.MACHINESTATE_Idle:
		bRed := FALSE;
		bGreen := FALSE;
		IF eSafetyState = E_SafetyState.Locked THEN
			bYellow := TRUE;
		ELSE
			bYellow := TRUE AND bBlink;
		END_IF
	ELSE
		bRed := FALSE;
		bYellow := FALSE;
		bGreen := TRUE AND bBlink;
END_CASE

ACTION A_Blink:
//Phase1
IF nStateBlink = 0 THEN
	bBlink := TRUE;
	tmrBlink(IN:= TRUE, PT:= T#1S);
	IF tmrBlink.Q THEN
		tmrBlink(IN:= FALSE);
		nStateBlink := 1;
	END_IF
END_IF

//Phase2
IF nStateBlink = 1 THEN
	bBlink := FALSE;
	tmrBlink(IN:= TRUE, PT:= T#1S);
	IF tmrBlink.Q THEN
		tmrBlink(IN:= FALSE);
		nStateBlink := 0;
	END_IF
END_IF
END_ACTION

END_FUNCTION_BLOCK

// ---- Hardware/Safety/FB_HwRefStopButton.TcPOU
FUNCTION_BLOCK FB_HwRefStopButton
VAR_INPUT
END_VAR
VAR_OUTPUT
END_VAR
VAR
	bE_Stop_NO 	AT %I* : BOOL;
	bE_Stop_NC 	AT %I* : BOOL;
	bRelease 	AT %Q* : BOOL; 
	bFTrig 		: F_TRIG;
END_VAR
VAR PERSISTENT
	bDisabled : BOOL := TRUE;
END_VAR

bRelease := NOT bE_Stop_NO AND bE_Stop_NC;
bFTrig(CLK:= (bRelease OR bDisabled));

PROPERTY P_bDisabled : BOOL
GET
P_bDisabled := bDisabled;
END_GET
SET
bDisabled := P_bDisabled;
fbSettings.M_WritePersData();
END_SET
END_PROPERTY

PROPERTY P_bReleased : BOOL
GET
P_bReleased := bRelease OR bDisabled;
END_GET
END_PROPERTY

PROPERTY P_bTriggered : BOOL
GET
P_bTriggered := bFTrig.Q;
END_GET
END_PROPERTY

END_FUNCTION_BLOCK

// ---- Hardware/Trigger/FB_TriggerOut.TcPOU
FUNCTION_BLOCK FB_TriggerOut
VAR_INPUT
END_VAR
VAR_OUTPUT
END_VAR
VAR
	//Start DS Änderung Plasmapen nur für 2372
	bPowerPlasma AT %Q*  	: BOOL;
	timer1					: TON;
	timer2					: TON;
	nState					: USINT := 0;
	// Ende
	bSafety AT %I* 	: BOOL;
	aOut AT %Q* 	: ARRAY[1..3] OF BOOL;
	aCycle			: ARRAY[1..3] OF USINT;
	i				: USINT;
END_VAR

//Wenn spätestens nach 2 Zyklen kein Ein mehr kommmt, dann ausschalten
FOR i:= 1 TO 3 BY 1 DO
	aCycle[i] := SHR(aCycle[i],1);
	aOut[i] := aCycle[i].0 AND bSafety;
END_FOR

//DS Änderung Plasmapen nur für 2372
timer1(PT:=T#5S);
timer2(PT:=T#2S);

CASE nState OF
	0:
	bPowerPlasma := TRUE;
	timer1(IN:=FALSE);
	timer2(IN:=FALSE);
	
	1:
	timer1(IN:=TRUE);
	IF timer1.Q THEN
		nState := 2;
	END_IF
	
	2:
	timer2(IN:=TRUE);
	bPowerPlasma := FALSE;
	IF timer2.Q THEN
		
		nState:=0;
		
	END_IF
	
END_CASE

METHOD FB_init : BOOL
VAR_INPUT
	bInitRetains : BOOL; // if TRUE, the retain variables are initialized (warm start / cold start)
	bInCopyCode : BOOL;  // if TRUE, the instance afterwards gets moved into the copy code (online change)
END_VAR
IF NOT (F_GetMappingStatus(ADR(bSafety),SIZEOF(bSafety)) = EPlcMappingStatus.MS_Partial) THEN
	bSafety := TRUE;
END_IF
END_METHOD

METHOD M_GetState : BOOL
VAR_INPUT
	nChannel : USINT;
END_VAR
IF nChannel >= 1 AND nChannel <= 3 THEN
	M_GetState := aOut[nChannel];
END_IF
END_METHOD

METHOD M_Off
VAR_INPUT
	nChannel : USINT;
END_VAR
IF nChannel >= 1 AND nChannel <= 3 THEN
	aCycle[nChannel] := 0;
	aOut[nChannel] := FALSE;
END_IF

	//DS Änderung Plasmapen nur für 2372
	nState:=1;
END_METHOD

METHOD M_On
VAR_INPUT
	nChannel : USINT;
END_VAR
IF nChannel >= 1 AND nChannel <= 3 THEN
	aCycle[nChannel] := 3;
END_IF

	//DS Änderung Plasmapen nur für 2372
	nState:=0;
END_METHOD

END_FUNCTION_BLOCK

// ---- Hardware/MultiZ/PWM/FB_MultiZPWM.TcPOU
FUNCTION_BLOCK FB_MultiZPWM
VAR_INPUT
END_VAR
VAR_OUTPUT
END_VAR
VAR
	bSafety AT %I* 	: BOOL;
	aEnable AT %Q* 	: ARRAY[1..2] OF USINT;
	aValue AT %Q* 	: ARRAY[1..2] OF UINT;
	aCycle			: ARRAY[1..3] OF USINT;
	i				: USINT;	
END_VAR

//Wenn spätestens nach 2 Zyklen kein Ein mehr kommmt, dann ausschalten
FOR i:= 1 TO 3 BY 1 DO
	aCycle[i] := SHR(aCycle[i],1);
	IF aCycle[i].0 AND bSafety THEN
		aEnable[i] := 1;
	ELSE
		aEnable[i] := 0;
	END_IF
END_FOR

METHOD FB_init : BOOL
VAR_INPUT
	bInitRetains : BOOL; // if TRUE, the retain variables are initialized (warm start / cold start)
	bInCopyCode : BOOL;  // if TRUE, the instance afterwards gets moved into the copy code (online change)
END_VAR
IF NOT (F_GetMappingStatus(ADR(bSafety),SIZEOF(bSafety)) = EPlcMappingStatus.MS_Partial) THEN
	bSafety := TRUE;
END_IF
END_METHOD

METHOD M_GetState : BOOL
VAR_INPUT
	nChannel : USINT;
END_VAR
IF nChannel >= 1 AND nChannel <= 2 THEN
	M_GetState := USINT_TO_BOOL(aEnable[nChannel]);
END_IF
END_METHOD

METHOD M_Off
VAR_INPUT
	nChannel : USINT;
END_VAR
IF nChannel >= 1 AND nChannel <= 2 THEN
	aCycle[nChannel] := 0;
	aEnable[nChannel] := 0;
	aValue[nChannel] := 0;
END_IF
END_METHOD

METHOD M_On
VAR_INPUT
	nChannel : USINT;
	nValue	 : UINT;	//Tastverhältnis in 1/10tel % 
END_VAR
//Wenn spätestens nach 2 Zyklen kein Ein mehr kommmt, dann ausschalten
IF nChannel >= 1 AND nChannel <= 2 THEN
	aCycle[nChannel] := 3;
	aValue[nChannel] := REAL_TO_UINT(1023.0 / 100.0 * (UINT_TO_REAL(nValue)/10.0));
END_IF
END_METHOD

END_FUNCTION_BLOCK

// ---- Hardware/XYDrive/FB_XYDrive_Lmt_DS.TcPOU
FUNCTION_BLOCK FB_XYDrive_Lmt_DS EXTENDS FB_XYDriveNC
VAR_INPUT
END_VAR
VAR_OUTPUT
END_VAR
VAR

	nCapturedCounter	AT %I* : UINT;
	nCapturedValue 		AT %I* : DINT;
	nErrorCode			AT %I* : UINT;
	nStatusWord			AT %I* : UINT;
	nCapturedCounterOld : UDINT;
	
	fbCoeWrite				: FB_EcCoESdoWrite;
	fbCoeRead				: FB_EcCoESdoRead;
	nCoeData				: DINT;
	//nCoeData16				: UINT;
	fbLmtChangePID			: FB_LmtChangePID;
	
	tmrHoming : TON;
	tmrTimeout : TON;
	
	nCycleCounter : USINT;
	
END_VAR

pAxisRefMaster^.ReadStatus();
rActPos := LREAL_TO_REAL(LIMIT(-999.0,pAxisRefMaster^.NcToPlc.ActPos,999.0) * 1000.0);

bHomed := pAxisRefMaster^.Status.Homed AND nStatusWord.11;

SUPER^();

//Falls Antrieb im Error steht (0x4650) den antriebssprzifischen Error auslesen
IF pAxisRefMaster^.Status.Error AND pAxisRefMaster^.Status.ErrorID = 16#4650 THEN
	stError.ErrorId := nErrorCode;
END_IF

ACTION A_Capture:
CASE nStateA_Capture OF
	0:	//Capture
		IF nCapturedCounter <> nCapturedCounterOld THEN
			IF eXYOrientation = E_XYOrientation.X THEN
				rCapturedPos := DINT_TO_REAL(nCapturedValue) / -10.0;
			ELSE
				rCapturedPos := DINT_TO_REAL(nCapturedValue) / 10.0;
			END_IF
			bCaptureOk := TRUE;
			nStateA_Capture := 80;
		END_IF
	70:
		nStateA_Capture := 80;
		bCaptureStopped := TRUE;
END_CASE
END_ACTION

ACTION A_Error:
IF nStateA_Error = 0 THEN
	IF nErrorId = 17744 OR nErrorId = 18000 THEN //Schleppabstandüberwachung "Position" bzw Antriebshardware nicht bereit
		nStateA_Error := 1;
	END_IF
END_IF

CASE nStateA_Error OF
	1:	//Achse ausschalten
		fbMcPower(Axis:= pAxisRefMaster^, Enable:= FALSE);
		IF NOT fbMcPower.Busy THEN
			nStateA_Error := 2;
		END_IF		
	
	2:	//Calibration zurücksetzen
		fbMcHome(Axis:= pAxisRefMaster^, Execute:= TRUE, HomingMode:= MC_ResetCalibration);
		IF NOT fbMcHome.Busy THEN
			IF fbMcHome.Error THEN
				nStateA_Error := 99;
			ELSE
				nStateA_Error := 3;
			END_IF
 			fbMcHome(Axis:= pAxisRefMaster^, Execute:= FALSE);
		END_IF
END_CASE
END_ACTION

ACTION A_Init:
CASE nStateA_Init OF
	0:	//DriveAdress der Achse ermitteln
		bBusy := TRUE;
		fbMcReadDriveAddress(Axis:= pAxisRefMaster^ ,Execute:= TRUE, DriveAddress=> stDriveAddress);
		IF NOT fbMcReadDriveAddress.Busy THEN
			IF fbMcReadDriveAddress.Error THEN
				nErrorId := UDINT_TO_UINT(fbMcReadDriveAddress.ErrorID);
				nStateA_Init := 99;
			ELSE
				nStateA_Init := 1;
			END_IF
			fbMcReadDriveAddress(Axis:= pAxisRefMaster^ ,Execute:= FALSE);
		END_IF

	1:	//Achse im Fehlerzustand?
		IF pAxisRefMaster^.Status.Error OR fbMcReset.Busy  THEN
			fbMcReset(Axis:= pAxisRefMaster^, Execute:= TRUE); 
			IF fbMcReset.Error THEN
				nErrorId := UDINT_TO_UINT(fbMcReset.ErrorID);
				fbMcReset(Axis:= pAxisRefMaster^, Execute := FALSE);
				nStateA_Init := 99;
			ELSIF fbMcReset.Done THEN
				fbMcReset(Axis:= pAxisRefMaster^, Execute := FALSE);
				nStateA_Init := 2;
			END_IF
		ELSE
			nStateA_Init := 2;
		END_IF
		
	2:	//Schleppabstandüberwachung deaktivieren
		fbMcWriteBoolParameter(Axis:= pAxisRefMaster^, Execute:= TRUE, ParameterNumber:= MC_AxisParameter.AxisEnPositionLagMonitoring, Value:= FALSE);
		IF NOT fbMcWriteBoolParameter.Busy THEN
			IF fbMcWriteBoolParameter.Error THEN
				nStateA_Init := 99;
			ELSE
				nStateA_Init := 3;
			END_IF
			fbMcWriteBoolParameter(Axis:= pAxisRefMaster^, Execute:= FALSE);
		END_IF
		
	3:	//NC "Referenziert-Flag" zurücksetzen
		fbMcHome(Axis:= pAxisRefMaster^, Execute:= TRUE, HomingMode:= MC_HomingMode.MC_ResetCalibration);
		IF NOT fbMcHome.Busy THEN
			fbMcHome(Axis:= pAxisRefMaster^, Execute:= FALSE);
			nStateA_Init := 4;
		END_IF
		
	4:	//NC "SoftEndlagenüberwachung "Min" deaktivieren
		fbMcWriteBoolParameter(Axis:= pAxisRefMaster^, Execute:= TRUE, ParameterNumber:= MC_AxisParameter.AxisEnMinSoftPosLimit, Value:= FALSE);
		IF NOT fbMcWriteBoolParameter.Busy THEN
			IF fbMcWriteBoolParameter.Error THEN
				nStateA_Init := 99;
			ELSE
				nStateA_Init := 5;
			END_IF
			fbMcWriteBoolParameter(Axis:= pAxisRefMaster^, Execute:= FALSE);
		END_IF

	5:	//NC "SoftEndlagenüberwachung "Max" deaktivieren
		fbMcWriteBoolParameter(Axis:= pAxisRefMaster^, Execute:= TRUE, ParameterNumber:= MC_AxisParameter.AxisEnMaxSoftPosLimit, Value:= FALSE);
		IF NOT fbMcWriteBoolParameter.Busy THEN
			IF fbMcWriteBoolParameter.Error THEN
				nStateA_Init := 99;
			ELSE
				nStateA_Init := 6;
			END_IF
			fbMcWriteBoolParameter(Axis:= pAxisRefMaster^, Execute:= FALSE);
		END_IF
	
	6:	//Achse freigegeben?
		IF bStop THEN
			fbMcPower(Axis:= pAxisRefMaster^, Enable:= FALSE);
			nStateA_Init := 80;
			RETURN;
		END_IF
		IF NOT pAxisRefMaster^.Status.ControlLoopClosed THEN
			fbMcPower(Axis:= pAxisRefMaster^, Enable:= TRUE, Enable_Positive:= TRUE, Enable_Negative:= TRUE, Override:= 100);
			IF fbMcPower.Error THEN
				nErrorId := UDINT_TO_UINT(fbMcPower.ErrorID);
				fbMcPower(Axis:= pAxisRefMaster^, Enable:= FALSE);
				nStateA_Init := 99;
			END_IF
		ELSE
			nStateA_Init := 7;
		END_IF
		
	7:	//Homing notwendig?
		IF NOT nStatusWord.11(*Homing Flag*) OR bReInit THEN
			IF bInvertInitDir THEN
				nCoeData := 16#A; //neg
			ELSE
				nCoeData := 16#B; //pos
			END_IF
			nStateA_Init := 8;
		ELSE
			nStateA_Init := 17;
		END_IF
		
	8:	//Homing-Richtung schreiben
		//Hier könnte es erforderlich sein, den Wert in dem ROM zu schreiben?
		fbCoeWrite(sNetId:= stDriveAddress.NetId, nSlaveAddr:= stDriveAddress.SlaveAddress, nIndex:= 16#2000 + 16#13C4, nSubIndex:= 1, 
				pSrcBuf:= ADR(nCoeData), cbBufLen:= SIZEOF(nCoeData), bExecute:= TRUE);
		IF NOT fbCoeWrite.bBusy THEN
			IF fbCoeWrite.bError THEN
				nStateA_Init := 99;
			ELSE
				nStateA_Init := 9;
				nCycleCounter := 0;
			END_IF
			fbCoeWrite(bExecute:= FALSE);
		END_IF		
	
	9:	//Home-Position schreiben
		IF eXYOrientation = E_XYOrientation.X THEN
			nCoeData := REAL_TO_DINT(rHomePos * -10.0);
		ELSE
			nCoeData := REAL_TO_DINT(rHomePos * 10.0);	
		END_IF
		nCycleCounter := nCycleCounter + 1;		
		fbCoeWrite(sNetId:= stDriveAddress.NetId, nSlaveAddr:= stDriveAddress.SlaveAddress, nIndex:= 16#2000 + 16#13C7, nSubIndex:= 1,
				pSrcBuf:= ADR(nCoeData), cbBufLen:= SIZEOF(nCoeData), bExecute:= TRUE);
		IF NOT fbCoeWrite.bBusy THEN
			IF fbCoeWrite.bError THEN
				nStateA_Init := 99;
			ELSE
				//SliderHomePos berechnen
				IF eXYOrientation = E_XYOrientation.X THEN
					nCoeData := REAL_TO_DINT(rHomePos * 10.0 + 378000.0);
				ELSE
					nCoeData := REAL_TO_DINT(rHomePos * 10.0 + 180000.0);	
				END_IF	
				nStateA_Init := 10;
			END_IF
			fbCoeWrite(bExecute:= FALSE);
		END_IF
		
	10:	//Slider-Home-Position schreiben
		fbCoeWrite(sNetId:= stDriveAddress.NetId, nSlaveAddr:= stDriveAddress.SlaveAddress, nIndex:= 16#2000 + 16#13CA, nSubIndex:= 1,
				pSrcBuf:= ADR(nCoeData), cbBufLen:= SIZEOF(nCoeData), bExecute:= TRUE);
		IF NOT fbCoeWrite.bBusy THEN
			IF fbCoeWrite.bError THEN
				nStateA_Init := 99;
			ELSE
				//nStateA_Init := 11;
				nStateA_Init := 20;
			END_IF
			fbCoeWrite(bExecute:= FALSE);
		END_IF
		
	20:	//PID-Parameter Regler modifizieren
		fbLmtChangePID(nMode:= 0, sNetId:= stDriveAddress.NetId, nSlaveAddr:= stDriveAddress.SlaveAddress, bExecute:= TRUE);
		IF NOT fbLmtChangePID.bBusy THEN
			IF fbLmtChangePID.bError THEN
				nStateA_Init := 99;
			ELSE
				nStateA_Init := 11;
			END_IF
			fbLmtChangePID(bExecute:= FALSE);
		END_IF
		
	11:	//Homig - Force mask setzen
		nCoeData := 1;
		fbCoeWrite(sNetId:= stDriveAddress.NetId, nSlaveAddr:= stDriveAddress.SlaveAddress, nIndex:= 16#2000 + 16#13F7, nSubIndex:= 1, 
				pSrcBuf:= ADR(nCoeData), cbBufLen:= SIZEOF(nCoeData), bExecute:= TRUE);
		IF NOT fbCoeWrite.bBusy THEN
			IF fbCoeWrite.bError THEN
				nStateA_Init := 99;
			ELSE
				nStateA_Init := 12;
			END_IF
			fbCoeWrite(bExecute:= FALSE);
		END_IF

	12:	//Homig - starten
		nCoeData := 1;
		fbCoeWrite(sNetId:= stDriveAddress.NetId, nSlaveAddr:= stDriveAddress.SlaveAddress, nIndex:= 16#2000 + 16#141F, nSubIndex:= 1, 
				pSrcBuf:= ADR(nCoeData), cbBufLen:= SIZEOF(nCoeData), bExecute:= TRUE);
		IF NOT fbCoeWrite.bBusy THEN
			IF fbCoeWrite.bError THEN
				nStateA_Init := 99;
			ELSE
				nStateA_Init := 13;
				tmrHoming(IN:= FALSE);				
			END_IF
			fbCoeWrite(bExecute:= FALSE);
		END_IF
		
	13:	//Homing state abrufen
		//Achse auf Error abfragen !!!
		IF bStop OR pAxisRefMaster^.Status.Error THEN
			fbMcPower(Axis:= pAxisRefMaster^, Enable:= FALSE);
			fbCoeRead(bExecute:= FALSE);
			nStateA_Init := 15;	//Stop Homing
			RETURN;
		END_IF
		tmrHoming(IN:= TRUE, PT:= T#100S);
		fbCoeRead(sNetId:= stDriveAddress.NetId, nSlaveAddr:= stDriveAddress.SlaveAddress, nIndex:= 16#2000 + 16#1B62, nSubIndex:= 1, 
				pDstBuf:= ADR(nCoeData), cbBufLen:= SIZEOF(nCoeData), bExecute:= TRUE);
		IF NOT fbCoeRead.bBusy THEN
			IF fbCoeRead.bError THEN
				nStateA_Init := 99;
			ELSE
				IF nCoeData = 16#090F THEN
					//nStateA_Init := 14;
					nStateA_Init := 21;
				END_IF
			END_IF
			fbCoeRead(bExecute:= FALSE);
		END_IF
		
	21:	//PID-Parameter Regler modifizieren
		fbLmtChangePID(nMode:= 1, sNetId:= stDriveAddress.NetId, nSlaveAddr:= stDriveAddress.SlaveAddress, bExecute:= TRUE);
		IF NOT fbLmtChangePID.bBusy THEN
			IF fbLmtChangePID.bError THEN
				nStateA_Init := 99;
			ELSE
				nStateA_Init := 14;
			END_IF
			fbLmtChangePID(bExecute:= FALSE);
		END_IF

		
	14:	//Warten, bis Position sich eingependelt
		Delay(IN:=TRUE , PT:=T#100MS);
		IF Delay.Q THEN
			Delay(IN:=FALSE);
			nStateA_Init := 15;
		END_IF

	15:	//Axis resetten, dadurch wird die Zielpos gleich der Istpos gesetzt
		fbMcReset(Axis:= pAxisRefMaster^, Execute:= TRUE);
		IF NOT fbMcReset.Busy THEN
			fbMcReset(Axis:= pAxisRefMaster^, Execute:= FALSE);
			nStateA_Init := 16;
		END_IF
		
	16:	//Homig - stoppen
		nCoeData := 0;
		fbCoeWrite(sNetId:= stDriveAddress.NetId, nSlaveAddr:= stDriveAddress.SlaveAddress, nIndex:= 16#2000 + 16#141F, nSubIndex:= 1, 
				pSrcBuf:= ADR(nCoeData), cbBufLen:= SIZEOF(nCoeData), bExecute:= TRUE);
		IF NOT fbCoeWrite.bBusy THEN
			IF fbCoeWrite.bError THEN
				nStateA_Init := 99;
			ELSE
				IF bStop OR pAxisRefMaster^.Status.Error THEN
					nStateA_Init := 18;
				ELSE
					nStateA_Init := 17;	
				END_IF
				
			END_IF
			fbCoeWrite(bExecute:= FALSE);
		END_IF
		
	17:	//NC "Referenziert-Flag" setzen
		fbMcHome(Axis:= pAxisRefMaster^, Execute:= TRUE, HomingMode:= MC_HomingMode.MC_ForceCalibration);
		IF NOT fbMcHome.Busy THEN
			fbMcHome(Axis:= pAxisRefMaster^, Execute:= FALSE);
			nStateA_Init := 18;
		END_IF
		
	18:	//NC "SoftEndlagenüberwachung "Min" aktivieren
		fbMcWriteBoolParameter(Axis:= pAxisRefMaster^, Execute:= TRUE, ParameterNumber:= MC_AxisParameter.AxisEnMinSoftPosLimit, Value:= TRUE);
		IF NOT fbMcWriteBoolParameter.Busy THEN
			IF fbMcWriteBoolParameter.Error THEN
				nStateA_Init := 99;
			ELSE
				nStateA_Init := 19;
			END_IF
			fbMcWriteBoolParameter(Axis:= pAxisRefMaster^, Execute:= FALSE);
		END_IF

	19:	//NC "SoftEndlagenüberwachung "Max" aktivieren
		fbMcWriteBoolParameter(Axis:= pAxisRefMaster^, Execute:= TRUE, ParameterNumber:= MC_AxisParameter.AxisEnMaxSoftPosLimit, Value:= TRUE);
		IF NOT fbMcWriteBoolParameter.Busy THEN
			IF fbMcWriteBoolParameter.Error THEN
				nStateA_Init := 99;
			ELSE
				IF pAxisRefMaster^.Status.Error THEN
					nStateA_Init := 99;
				ELSE
					nStateA_Init := 80;
				END_IF
				
			END_IF
			fbMcWriteBoolParameter(Axis:= pAxisRefMaster^, Execute:= FALSE);
		END_IF
		
	99:	//Error
		fbMcPower(Axis:= pAxisRefMaster^, Enable:= FALSE);
		bError := TRUE;
END_CASE
END_ACTION

ACTION A_Reset:

CASE nStateA_Reset OF
	0:	
		bBusy := TRUE;
		IF pAxisRefMaster^.Status.Error THEN
			IF pAxisRefMaster^.Status.ErrorID = 16#4550 OR pAxisRefMaster^.Status.ErrorID = 16#4650 THEN
				//16#4550 Schleppabstand, 16#4650 Antriebshardware nicht bereit
				nStateA_Reset := 1;
			ELSIF pAxisRefMaster^.Status.ErrorID = 16#4655 THEN //ungültige Daten (eventuell durch Resetting von anderem Device)
				//warten bis WcState wieder "0" mit max. Timeout 15s
				IF pAxisRefMaster^.Status.IoDataInvalid THEN
					tmrTimeout(IN:= TRUE, PT:= T#15S);
					IF tmrTimeout.Q THEN
						tmrTimeout(IN:= FALSE);
						nStateA_Reset := 99;
					END_IF
				ELSE
					tmrTimeout(IN:= FALSE);
					nStateA_Reset := 4;	
				END_IF
			ELSE
				nStateA_Reset := 4;
			END_IF
		ELSE
			nStateA_Reset := 5;
		END_IF
	
	1:	//Reset Calibration
		fbMcHome(Axis:= pAxisRefMaster^, Execute:= TRUE, HomingMode:= Tc2_MC2.MC_HomingMode.MC_ResetCalibration);
		IF NOT fbMcHome.Busy THEN
			fbMcHome(Axis:= pAxisRefMaster^, Execute:= FALSE);
			nStateA_Reset := 2;
		END_IF
		
	2:	IF pAxisRefMaster^.Status.ErrorID = 16#4650 THEN //Antriebshardware nicht bereit -> Drive zurcüksetzen
			fbCoeWrite(sNetId:= stAdsAddress.sNetId, nSlaveAddr:= stAdsAddress.nPort, nIndex:= 16#2000, nSubIndex:= 16#0B,
					pSrcBuf:= ADR(nCoeData), cbBufLen:= 0, tTimeout := T#10S, bExecute:= TRUE);
			IF NOT fbCoeWrite.bBusy THEN
				IF fbCoeWrite.bError THEN
					nStateA_Reset := 99;
				ELSE
					tmrTimeout(IN:= TRUE, PT:= T#15S); //Achse sollte sich spätestens nach 15sec. wieder melden
					nStateA_Reset := 3;
				END_IF
				fbCoeWrite(bExecute:= FALSE);
			END_IF
			
		END_IF
		
	3:	//Fehler zurückgesetzt?
		tmrTimeout();
		IF tmrTimeout.Q THEN
			tmrTimeout(IN:= FALSE);
			nStateA_Reset := 99;
		END_IF
		
		IF nErrorCode = 0 THEN
			tmrTimeout(IN:= FALSE);
			nStateA_Reset := 4;
		END_IF
	
	4:	//Reset NC Achse
		fbMcReset(Axis:= pAxisRefMaster^, Execute:= TRUE);
		IF NOT fbMcReset.Busy THEN
			fbMcReset(Axis:= pAxisRefMaster^, Execute:= FALSE);
			nStateA_Reset := 5;
		END_IF
	
	5:	//Checken, ob Achse fehlerfrei
		IF pAxisRefMaster^.Status.Error THEN
			nStateA_Reset := 99;
		ELSE
			//Motion-Bausteine zurücksetzen
			fbMcMoveAbs(Axis:= pAxisRefMaster^, Execute:= FALSE);
			fbMcMoveRel(Axis:= pAxisRefMaster^, Execute:= FALSE);
			fbMcHalt(Axis:= pAxisRefMaster^, Execute:= FALSE);
			nStateA_Reset := 80;
			nStateA_Error := 0;
			bError := FALSE;
		END_IF
END_CASE
END_ACTION

ACTION A_Setup:
CASE nStateA_Setup OF
	0:	//Achsen initialisieren mit RefPos0 (RefPos0 wird in M_Setup() gesetzt
		bInit := TRUE;
		nStateA_Setup := 1;
		bSetupWaitForResp := FALSE;
		
	1:	//Warten bis "Init" fertig"
		IF NOT bInit THEN
			nStateA_Setup := 2;
		END_IF

	2:	//Homed zurücksetzen durch die nächsten 3 Steps
		//HomingSpeed auf "0" setzen
		nCoeData := 0;
		fbCoeWrite(sNetId:= stDriveAddress.NetId, nSlaveAddr:= stDriveAddress.SlaveAddress, nIndex:= 16#2000 + 16#13C8, nSubIndex:= 1, 
				pSrcBuf:= ADR(nCoeData), cbBufLen:= SIZEOF(nCoeData), bExecute:= TRUE);
		IF NOT fbCoeWrite.bBusy THEN
			IF fbCoeWrite.bError THEN
				nStateA_Setup := 99;
			ELSE
				nStateA_Setup := 3;
			END_IF
			fbCoeWrite(bExecute:= FALSE);
		END_IF
		
	3:	//Homing starten
		nCoeData := 1;
		fbCoeWrite(sNetId:= stDriveAddress.NetId, nSlaveAddr:= stDriveAddress.SlaveAddress, nIndex:= 16#2000 + 16#141F, nSubIndex:= 1, 
				pSrcBuf:= ADR(nCoeData), cbBufLen:= SIZEOF(nCoeData), bExecute:= TRUE);
		IF NOT fbCoeWrite.bBusy THEN
			IF fbCoeWrite.bError THEN
				nStateA_Setup := 99;
			ELSE
				nStateA_Setup := 4;
			END_IF
			fbCoeWrite(bExecute:= FALSE);
		END_IF
		
	4:	//Homing stoppen
		nCoeData := 0;
		fbCoeWrite(sNetId:= stDriveAddress.NetId, nSlaveAddr:= stDriveAddress.SlaveAddress, nIndex:= 16#2000 + 16#141F, nSubIndex:= 1, 
				pSrcBuf:= ADR(nCoeData), cbBufLen:= SIZEOF(nCoeData), bExecute:= TRUE);
		IF NOT fbCoeWrite.bBusy THEN
			IF fbCoeWrite.bError THEN
				nStateA_Setup := 99;
			ELSE
				nStateA_Setup := 5;
			END_IF
			fbCoeWrite(bExecute:= FALSE);
		END_IF
		
	5:	//HomingSpeed auf "0.02" setzen
		nCoeData := 20000;
		fbCoeWrite(sNetId:= stDriveAddress.NetId, nSlaveAddr:= stDriveAddress.SlaveAddress, nIndex:= 16#2000 + 16#13C8, nSubIndex:= 1, 
				pSrcBuf:= ADR(nCoeData), cbBufLen:= SIZEOF(nCoeData), bExecute:= TRUE);
		IF NOT fbCoeWrite.bBusy THEN
			IF fbCoeWrite.bError THEN
				nStateA_Setup := 99;
			ELSE
				nStateA_Setup := 6;
			END_IF
			fbCoeWrite(bExecute:= FALSE);
		END_IF
		
	6:	//Achse ausschalten
		fbMcPower(Axis:= pAxisRefMaster^, Enable:= FALSE);
		IF NOT pAxisRefMaster^.Status.ControlLoopClosed THEN
			IF bStop THEN
				nStateA_Setup := 80;
			ELSE
				nStateA_Setup := 10; //Weiterschalten zu "11" werfolgt durch fbConfigSetup
				bSetupWaitForResp := TRUE; //Wartet auf Antwort vom User
				bContinueSetup := FALSE;
			END_IF
		END_IF
		
	10:	//Warte auf UserResponse
		IF bStop THEN
			nStateA_Setup := 80;
		ELSE
			IF bContinueSetup THEN
				nStateA_Setup := 11;
			END_IF
		END_IF
		
	11:	//Referenzposition berechnen
		IF eXYOrientation = E_XYOrientation.X THEN
			rRefPosMaster := rWorkplateLength - rActPos - rSetupPosDist - rNullPosDist;
		ELSE
			rRefPosMaster := (-rActPos) + rSetupPosDist - rNullPosDist;
		END_IF
		nStateA_Setup := 80;
	
END_CASE
END_ACTION

ACTION A_StopCapture:
CASE nStateA_StopCapture OF
	0:	IF bCapture AND nStateA_Capture < 70 THEN
			nStateA_Capture := 70;
			nStateA_StopCapture := 1;
		ELSE
			nStateA_StopCapture := 80;
		END_IF
		
	1:	IF NOT bCapture THEN
			bCaptureStopped := TRUE;
			nStateA_StopCapture := 80;
		END_IF
END_CASE
END_ACTION

ACTION A_WriteAxisParameter:
IF nStateA_WriteAxisParamter = 0 THEN
	//feststellen, welcher Parameter als nächstes geschrieben werden muss
	IF nStateWriteLimitNegative = 1 THEN
		nStateWriteLimitNegative := 2;
	ELSIF nStateWriteLimitPositive = 1 THEN
		nStateWriteLimitPositive := 2;
	ELSIF nStateWriteNCIFastSpeed = 1 THEN
		nStateWriteNCIFastSpeed := 2;
	ELSE
		nStateWriteLimitNegative := 1;
		nStateWriteLimitPositive := 1;
		nStateWriteNCIFastSpeed := 1;
		nStateA_WriteAxisParamter := 80;
		RETURN;
	END_IF
	
	IF nStateWriteLimitNegative = 2 THEN
		fbMcWriteParameter.ParameterNumber := MC_AxisParameter.SWLimitNeg;
		fbMcWriteParameter.Value := P_rMinPos / 1000.0;
		nStateA_WriteAxisParamter := 1;
	END_IF
	
	IF nStateWriteLimitPositive = 2 THEN
		fbMcWriteParameter.ParameterNumber := MC_AxisParameter.SWLimitPos;
		fbMcWriteParameter.Value := P_rMaxPos / 1000.0;
		nStateA_WriteAxisParamter := 1;
	END_IF

	IF nStateWriteNCIFastSpeed = 2 THEN
		fbMcWriteParameter.ParameterNumber := MC_AxisParameter.AxisRapidTraverseVelocity;
		fbMcWriteParameter.Value := rMaxSpeed / 1000.0;
		nStateA_WriteAxisParamter := 1;
	END_IF
	
END_IF

IF nStateA_WriteAxisParamter = 1 THEN
	fbMcWriteParameter(Axis:= pAxisRefMaster^, Execute:= TRUE);
	//Hier kann es passieren, dass der Fehler "1793" auftritt. Das passiert manchmal beim Start der SPS
	//In diesem Falle, sollte es solange probiert werden, bis dieser nicht mehr auftritt
	IF NOT fbMcWriteParameter.Busy THEN
		IF fbMcWriteParameter.Error THEN
			IF fbMcWriteParameter.ErrorID <> 1793 THEN
				nStateA_WriteAxisParamter := 99;
			END_IF
		ELSE
			CASE fbMcWriteParameter.ParameterNumber OF
				MC_AxisParameter.SWLimitNeg:
					nStateWriteLimitNegative := 3;
				MC_AxisParameter.SWLimitPos:
					nStateWriteLimitPositive := 3;
				MC_AxisParameter.AxisRapidTraverseVelocity:
					nStateWriteNCIFastSpeed := 3;
			END_CASE
			nStateA_WriteAxisParamter := 0;
		END_IF
		fbMcWriteParameter(Axis:= pAxisRefMaster^, Execute:= FALSE);
	END_IF	
END_IF
END_ACTION

METHOD FB_init : BOOL
VAR_INPUT
	bInitRetains 	: BOOL; // if TRUE, the retain variables are initialized (warm start / cold start)
	bInCopyCode 	: BOOL;  // if TRUE, the instance afterwards gets moved into the copy code (online change)
	eXYOrientation	: E_XYOrientation;
	pNCAxisRef		: POINTER TO AXIS_REF;
END_VAR
THIS^.pAxisRefMaster := pNCAxisRef;
END_METHOD

METHOD M_Capture : ERRORID
VAR_INPUT
END_VAR
nCapturedCounterOld := nCapturedCounter;
bCapture := TRUE;
bCaptureOk := FALSE;
bCaptureStopped := FALSE;
A_Capture();
END_METHOD

PROPERTY P_bHasJob : BOOL
GET
pAxisRefMaster^.ReadStatus();
P_bHasJob := pAxisRefMaster^.Status.HasJob;
END_GET
END_PROPERTY

PROPERTY P_bIsMoving : BOOL
GET
pAxisRefMaster^.ReadStatus();
P_bIsMoving :=  pAxisRefMaster^.Status.Moving;
END_GET
END_PROPERTY

PROPERTY P_pAxisRef : POINTER TO AXIS_REF
GET
P_pAxisRef := pAxisRefMaster;
END_GET
END_PROPERTY

PROPERTY P_tHomingTime : TIME
GET
P_tHomingTime := tmrHoming.ET;
END_GET
END_PROPERTY

END_FUNCTION_BLOCK

// ---- Hardware/XYDrive/FB_LmtChangePID.TcPOU
FUNCTION_BLOCK FB_LmtChangePID
VAR_INPUT
	nMode		: USINT; //0= B_ROM_To_A_RAM ;  1= A_ROM_TO_A_RAM
	sNetId 		: T_AmsNetID;
	nSlaveAddr 	: UINT;
	bExecute	: BOOL;
END_VAR
VAR_OUTPUT
	bBusy : BOOL;
	bError : BOOL;
END_VAR
VAR
	nState 		: USINT;
	nStateAct	: USINT;
	fbCoeWrite	: FB_EcCoESdoWrite;
	fbCoeRead	: FB_EcCoESdoRead;
	
	nPGainRomA : DINT;
	nDGainRomA : DINT;
	nIGainRomA : DINT;
	nPGainRomB : DINT;
	nDGainRomB : DINT;
	nIGainRomB : DINT;
	nPGainRamA : DINT;
	nDGainRamA : DINT;	
	nIGainRamA : DINT;
	
	nStep : USINT;
	nPGainIncreaseValue : DINT;
	nDGainIncreaseValue : DINT;
	nIGainIncreaseValue : DINT;
	
END_VAR

//Dient zum Anpassen der aktuellen ParameterA im RAM
IF bExecute THEN
	bBusy := TRUE;

	IF nState = 0 THEN	//Read ROM B
		A_ReadRomB();
		IF nStateAct >= 80 THEN
			IF nStateAct >= 99 THEN
				nState := 99;
			ELSE
				IF nMode = 0 THEN
					nPGainRamA := nPGainRomB;
					nDGainRamA := nDGainRomB;
					nIGainRamA := nIGainRomB;
					nState := 3;
				ELSE
					nState := 1;
				END_IF
			END_IF
			nStateAct := 0;
		END_IF
	END_IF

	IF nState = 1 THEN	//Read ROM A
		A_ReadRomA();
		IF nStateAct >= 80 THEN
			IF nStateAct >= 99 THEN
				nState := 99;
			ELSE
				nStep := 0;
				nPGainIncreaseValue := (nPGainRomA - nPGainRomB) / 10;
				nDGainIncreaseValue := (nDGainRomA - nDGainRomB) / 10;
				nIGainIncreaseValue := (nIGainRomA - nIGainRomB) / 10;
				nPGainRamA := nPGainRomB;
				nDGainRamA := nDGainRomB;
				nIGainRamA := nIGainRomB;
				
				nState := 2;
			END_IF
			nStateAct := 0;
		END_IF
	END_IF
	
	IF nState = 2 THEN	//Increase
		nStep := nStep + 1;
		nPGainRamA := MIN(nPGainRomA,nPGainRamA + nPGainIncreaseValue);
		nDGainRamA := MIN(nDGainRomA,nDGainRamA + nDGainIncreaseValue);
		nIGainRamA := MIN(nIGainRomA,nIGainRamA + nPGainIncreaseValue);
		nState := 3;
	END_IF
	
	IF nState = 3 THEN	//Write ROM A
		A_WriteRamA();
		IF nStateAct >= 80 THEN
			IF nStateAct >= 99 THEN
				nState := 99;
			ELSE
				IF nMode = 0 THEN
					nState := 80;
				ELSIF nMode = 1 THEN
					IF nPGainRomA = nPGainRamA AND nDGainRomA = nDGainRamA AND nIGainRomA = nIGainRamA THEN
						nState := 80;
					ELSE
						nState := 2; //Increase
					END_IF
				END_IF
			END_IF
			nStateAct := 0;
		END_IF
	END_IF

	IF nState >= 80 THEN
		IF nState >= 99 THEN
			bError := TRUE;			
		END_IF
		bBusy := FALSE;
	END_IF

ELSE
	nState := 0;
	nStateAct := 0;
	bError := FALSE;
	fbCoeRead(bExecute:= FALSE);
	fbCoeWrite(bExecute:= FALSE);
END_IF

ACTION A_ReadRomA:
IF nStateAct = 0 THEN	//PGain
	fbCoeRead(sNetId:= sNetId, nSlaveAddr:= nSlaveAddr, nIndex:= 16#2000 + 16#13A2, nSubIndex:= 2(*Read Rom = 2*), 
			pDstBuf:= ADR(nPGainRomA), cbBufLen:= SIZEOF(nPGainRomB), bExecute:= TRUE);
	IF NOT fbCoeRead.bBusy THEN
		IF fbCoeRead.bError THEN
			nStateAct := 99;
		ELSE
			nStateAct := 1;
		END_IF
		fbCoeRead(bExecute:= FALSE);
	END_IF			
END_IF

IF nStateAct = 1 THEN	//DGain
	fbCoeRead(sNetId:= sNetId, nSlaveAddr:= nSlaveAddr, nIndex:= 16#2000 + 16#13A3, nSubIndex:= 2(*Read Rom = 2*), 
			pDstBuf:= ADR(nDGainRomA), cbBufLen:= SIZEOF(nDGainRomB), bExecute:= TRUE);
	IF NOT fbCoeRead.bBusy THEN
		IF fbCoeRead.bError THEN
			nStateAct := 99;
		ELSE
			nStateAct := 2;
		END_IF
		fbCoeRead(bExecute:= FALSE);
	END_IF		
END_IF

IF nStateAct = 2 THEN	//IGain
	fbCoeRead(sNetId:= sNetId, nSlaveAddr:= nSlaveAddr, nIndex:= 16#2000 + 16#13A4, nSubIndex:= 2(*Read Rom = 2*), 
			pDstBuf:= ADR(nIGainRomA), cbBufLen:= SIZEOF(nIGainRomB), bExecute:= TRUE);
	IF NOT fbCoeRead.bBusy THEN
		IF fbCoeRead.bError THEN
			nStateAct := 99;
		ELSE
			nStateAct := 80;
		END_IF
		fbCoeRead(bExecute:= FALSE);
	END_IF		
END_IF
END_ACTION

ACTION A_ReadRomB:
IF nStateAct = 0 THEN	//PGain
	fbCoeRead(sNetId:= sNetId, nSlaveAddr:= nSlaveAddr, nIndex:= 16#2000 + 16#13B6, nSubIndex:= 2(*Read Rom = 2*), 
			pDstBuf:= ADR(nPGainRomB), cbBufLen:= SIZEOF(nPGainRomB), bExecute:= TRUE);
	IF NOT fbCoeRead.bBusy THEN
		IF fbCoeRead.bError THEN
			nStateAct := 99;
		ELSE
			nStateAct := 1;
		END_IF
		fbCoeRead(bExecute:= FALSE);
	END_IF			
END_IF

IF nStateAct = 1 THEN	//DGain
	fbCoeRead(sNetId:= sNetId, nSlaveAddr:= nSlaveAddr, nIndex:= 16#2000 + 16#13B7, nSubIndex:= 2(*Read Rom = 2*), 
			pDstBuf:= ADR(nDGainRomB), cbBufLen:= SIZEOF(nDGainRomB), bExecute:= TRUE);
	IF NOT fbCoeRead.bBusy THEN
		IF fbCoeRead.bError THEN
			nStateAct := 99;
		ELSE
			nStateAct := 2;
		END_IF
		fbCoeRead(bExecute:= FALSE);
	END_IF		
END_IF

IF nStateAct = 2 THEN	//IGain
	fbCoeRead(sNetId:= sNetId, nSlaveAddr:= nSlaveAddr, nIndex:= 16#2000 + 16#13B8, nSubIndex:= 2(*Read Rom = 2*), 
			pDstBuf:= ADR(nIGainRomB), cbBufLen:= SIZEOF(nIGainRomB), bExecute:= TRUE);
	IF NOT fbCoeRead.bBusy THEN
		IF fbCoeRead.bError THEN
			nStateAct := 99;
		ELSE
			nStateAct := 80;
		END_IF
		fbCoeRead(bExecute:= FALSE);
	END_IF		
END_IF
END_ACTION

ACTION A_WriteRamA:
IF nStateAct = 0 THEN	//PGain
	fbCoeWrite(sNetId:= sNetId, nSlaveAddr:= nSlaveAddr, nIndex:= 16#2000 + 16#13A2, nSubIndex:= 1(*1=RAM*), 
			pSrcBuf:= ADR(nPGainRamA), cbBufLen:= SIZEOF(nPGainRamA), bExecute:= TRUE);
	IF NOT fbCoeWrite.bBusy THEN
		IF fbCoeWrite.bError THEN
			nStateAct := 99;
		ELSE
			nStateAct := 1;
		END_IF
		fbCoeWrite(bExecute:= FALSE);
	END_IF	
END_IF

IF nStateAct = 1 THEN	//DGain
	fbCoeWrite(sNetId:= sNetId, nSlaveAddr:= nSlaveAddr, nIndex:= 16#2000 + 16#13A3, nSubIndex:= 1(*1=RAM*), 
			pSrcBuf:= ADR(nDGainRamA), cbBufLen:= SIZEOF(nDGainRamA), bExecute:= TRUE);
	IF NOT fbCoeWrite.bBusy THEN
		IF fbCoeWrite.bError THEN
			nStateAct := 99;
		ELSE
			nStateAct := 2;
		END_IF
		fbCoeWrite(bExecute:= FALSE);
	END_IF	
END_IF

IF nStateAct = 2 THEN	//IGain
	fbCoeWrite(sNetId:= sNetId, nSlaveAddr:= nSlaveAddr, nIndex:= 16#2000 + 16#13A4, nSubIndex:= 1(*1=RAM*), 
			pSrcBuf:= ADR(nIGainRamA), cbBufLen:= SIZEOF(nIGainRamA), bExecute:= TRUE);
	IF NOT fbCoeWrite.bBusy THEN
		IF fbCoeWrite.bError THEN
			nStateAct := 99;
		ELSE
			nStateAct := 80;
		END_IF
		fbCoeWrite(bExecute:= FALSE);
	END_IF	
END_IF
END_ACTION

END_FUNCTION_BLOCK

// ---- Hardware/XYDrive/FB_XYDrive_Lmt_EC.TcPOU
FUNCTION_BLOCK FB_XYDrive_Lmt_EC EXTENDS FB_XYDriveBase
VAR_INPUT
END_VAR
VAR_OUTPUT
END_VAR
VAR
	
	bPowerOn : BOOL;
	nStateA_PowerOn : USINT;
	timeout	: TON;
	
	tmrHoming	: TON;

	nCapturedCounter	AT %I* : UINT;
	nCapturedValue 		AT %I* : DINT;
	nCapturedCounterOld : UDINT;
	
	fbAxisControl 		: Tc3_LinMot.LMct_AxisControl;
	fbLMcfParaAccess 	: Tc3_LinMot.LMcf_ParaAccess;
	fbLMmtMoveRel		: Tc3_LinMot.LMmt_MoveRel;
	fbLMmtMoveAbs		: Tc3_LinMot.LMmt_MoveAbs;
	fbLMmtStop			: Tc3_Linmot.LMmt_Stop;
	fbCoeWrite			: FB_EcCoESdoWrite;
	nCoeData			: DINT;
	
	rSliderHomePos : REAL;
	
	pAxisRef : POINTER TO Tc3_LinMot.tstLM_Axis;
END_VAR

SUPER^();
fbAxisControl(Axis:= pAxisRef^);
rActPos := fbAxisControl.ActualPosition * 1000.0;
bHomed := fbAxisControl.Homed;
bError := fbAxisControl.Error;
nErrorId := fbAxisControl.ErrorCode + 42751;

fbLMmtStop(Axis:= pAxisRef^);
IF NOT fbLMmtStop.Busy THEN
	fbLMmtStop(Axis:= pAxisRef^, Execute:= FALSE);
END_IF

IF bPowerOn THEN
	A_PowerOn();
	IF nStateA_PowerOn >= 80 THEN
		IF nStateA_PowerOn >= 99 THEN
			bError := TRUE;
		END_IF
		nStateA_PowerOn := 0;
		bPowerOn := FALSE;
	END_IF
END_IF

bBusy := bBusy OR bPowerOn;

ACTION A_PowerOn:
timeout();
IF timeout.Q THEN
	timeout(IN:= FALSE);
	fbAxisControl(ErrorAcknowledge := FALSE, SwitchOn := FALSE, JogPlus:= FALSE, JogMinus:= FALSE, Home:= FALSE, Axis:= pAxisRef^);
	nStateA_PowerOn := 99;
	bError := TRUE;
	bBusy := FALSE;
END_IF

IF nStateA_PowerOn = 0 THEN //Achse im Fehlerzustand?
	IF fbAxisControl.Error THEN
		timeout(IN:= TRUE, PT:= T#5S);
		fbAxisControl(ErrorAcknowledge := TRUE, SwitchOn := FALSE, JogPlus:= FALSE, JogMinus:= FALSE, Home:= FALSE, Axis:= pAxisRef^);
	ELSE
		timeout(IN:= FALSE);
		fbAxisControl.ErrorAcknowledge := FALSE;
		nStateA_PowerOn := 1;
	END_IF	
END_IF

IF nStateA_PowerOn = 1 THEN //Achse einschalten
	timeout(IN:= TRUE, PT:= T#3S);
	fbAxisControl(SwitchOn := TRUE,JogPlus:= FALSE, JogMinus:= FALSE, Axis:= pAxisRef^);
	IF fbAxisControl.OperationEnabled THEN
		timeout(IN:= FALSE);
		nStateA_PowerOn := 80;
	END_IF
END_IF
END_ACTION

ACTION A_MoveRel:
IF fbLMmtMoveRel.Error THEN
	nErrorId := UDINT_TO_UINT(fbLMmtMoveRel.ErrorId);
	fbLMmtMoveRel(Axis:= pAxisRef^, Execute:= FALSE);
	nStateMoveRel := 99;
END_IF

CASE nStateMoveRel OF
	0:	IF bStop THEN
			nStateMoveRel := 80;
		ELSE
			bBusy := TRUE;
			fbLMmtMoveRel(Axis:= pAxisRef^, Execute:= TRUE);
			nStateMoveRel := 1;
		END_IF
	
	1:	//Warten bis Move fertig
		IF bStop THEN
			fbLMmtStop(Execute:= TRUE, Axis:= pAxisRef^, Deceleration:= 1.0);
			fbLMmtMoveRel(Axis:= pAxisRef^, Execute:= FALSE);
			nStateMoveRel := 2;		
		ELSE
			fbLMmtMoveRel(Axis:= pAxisRef^);
			IF NOT fbLMmtMoveRel.Busy THEN
				fbLMmtMoveRel(Axis:= pAxisRef^, Execute:= FALSE);
				nStateMoveRel := 80;
			END_IF
		END_IF
		
	2:	//Warten bis Stop fertig
		IF fbLMmtStop.Error THEN
			bError := TRUE;
			nErrorId := fbLMmtStop.ErrorID;
			nStateMoveRel := 99;
			bStop := FALSE;
		END_IF
		
		IF NOT fbLMmtStop.Busy THEN
			fbLMmtStop(Execute:= FALSE, Axis:= pAxisRef^);
			nStateMoveRel := 80;
			bStop := FALSE;
		END_IF	
END_CASE
END_ACTION

ACTION A_Capture:
CASE nStateA_Capture OF
	0:	//Capture
		IF nCapturedCounter <> nCapturedCounterOld THEN
			IF eXYOrientation = E_XYOrientation.X THEN
				rCapturedPos := DINT_TO_REAL(nCapturedValue) / -10.0;
			ELSE
				rCapturedPos := DINT_TO_REAL(nCapturedValue) / 10.0;
			END_IF
			bCaptureOk := TRUE;
			nStateA_Capture := 80;
		END_IF
	70:
		nStateA_Capture := 80;
		
END_CASE
END_ACTION

METHOD M_PowerOn : ERRORID
VAR_INPUT
END_VAR
bPowerOn := TRUE;
END_METHOD

METHOD M_Jog : ERRORID
VAR_INPUT
	bForward	: BOOL;
	bBackward	: BOOL;
	bInching	: BOOL;
	rDistance	: REAL;
	rSpeed		: REAL;	
END_VAR
IF bInching THEN
	//Hier müssen auch die Grenzen gecheckt werden!!
	IF (bBackward AND eXYOrientation = E_XYOrientation.Y) OR (NOT bBackward AND eXYOrientation = E_XYOrientation.X) THEN
		rDistance := rDistance * -1.0;
	END_IF
	fbLMmtMoveRel.Distance := rDistance / 1000.0;
	fbLMmtMoveRel.Velocity := rSpeed / 1000000.0;
	fbLMmtMoveRel.Acceleration := 1.0;
	fbLMmtMoveRel.Deceleration := 1.0;
ELSE //Conti
	//Die Position muss aus den maximalen Grenzen ermittelt werden!!
	IF bForward THEN
		fbLMmtMoveAbs.Position := P_rMaxPos / 1000.0;
	ELSIF bBackward THEN
		fbLMmtMoveAbs.Position := P_rMinPos / 1000.0;
	END_IF
	
	IF eXYOrientation = E_XYOrientation.X THEN
		fbLMmtMoveAbs.Position := fbLMmtMoveAbs.Position * -1.0;
	END_IF
	
	fbLMmtMoveAbs.Velocity := rSpeed / 1000000.0;
	fbLMmtMoveAbs.Acceleration := 1.0;
	fbLMmtMoveAbs.Deceleration := 1.0;
END_IF

//Ein Richtungswechsel bzw. Modewechsel sollte immer erst einen Stop ausführen, falls Jog noch aktiv ist.
IF bJog THEN
	IF bForward <> bJogForward OR bBackward <> bJogBackward OR bInching <> bJogInching THEN
		//Stoppen und falls kein Stop angefordert, dann neu mit neuen Paramtern ausführen
		//für diesen Fall müssen die Parameter zwischengespeichert werden?
		nStateA_Jog := 70;
		A_Jog();
		bJogForward := bForward;
		bJogBackward := bBackward;
		bJogInching := bInching;		
	ELSE
		//continuierliches Joggen:
		//Timer zurücksetzen und nStateA_Jog auf "0" setzen
		//inkrementelles Joggen wird nicht erneut angenommen, wenn es bereits aktiv ist und die gleichen Paramter aufweist
		IF NOT bJogInching THEN
			tmrJog(IN:=FALSE);
			nStateA_Jog := 0;
			A_Jog();			
		END_IF
	END_IF
ELSE
	IF bBusy THEN
		M_Jog := 23244;
	ELSE
		bJog := TRUE;
		bJogForward := bForward;
		bJogBackward := bBackward;
		bJogInching := bInching;		
		A_Jog();
	END_IF
END_IF
END_METHOD

METHOD FB_init : BOOL
VAR_INPUT
	bInitRetains 	: BOOL; // if TRUE, the retain variables are initialized (warm start / cold start)
	bInCopyCode 	: BOOL;  // if TRUE, the instance afterwards gets moved into the copy code (online change)
	eXYOrientation	: E_XYOrientation;
	pAxisRef		: POINTER TO Tc3_LinMot.tstLM_Axis;		
END_VAR
THIS^.pAxisRef := pAxisRef;
END_METHOD

PROPERTY P_rActPos : REAL
GET
IF eXYOrientation = E_XYOrientation.X THEN
	P_rActPos := rActPos * -1.0;
ELSE
	P_rActPos := rActPos;	
END_IF
END_GET
END_PROPERTY

ACTION A_Setup:
CASE nStateA_Setup OF
	0:	//Achsen initialisieren mit RefPos0
		bInit := TRUE;
		nStateA_Setup := 1;
		bSetupWaitForResp := FALSE;
		
	1:	//Warten bis "Init" fertig"
		IF NOT bInit THEN
			nStateA_Setup := 2;
		END_IF
		
		IF bStop THEN
			nStateA_Setup := 80;
		END_IF
 
		
	2:	//HomingSpeed auf "0" setzen, damit Antrieb nicht mehr "Homed"
		fbLMcfParaAccess(Execute:= TRUE , Mode:= 3, UPIDIn:=16#13C8 , Axis:= pAxisRef^, ValueIn := 0);
		IF NOT fbLMcfParaAccess.Busy THEN
			IF fbLMcfParaAccess.Error THEN
				nErrorId := fbLMcfParaAccess.ErrorID;
				nStateA_Setup := 99;
			ELSE
				nStateA_Setup := 3;	
			END_IF
			fbLMcfParaAccess(Execute:= FALSE, Axis:= pAxisRef^);
		END_IF
		
	3:	//Homing erneut starten
		fbAxisControl(Home := TRUE, Axis:= pAxisRef^);
		IF pAxisRef^.AxisState = tenLM_AxisState.Homing_LM THEN
			nStateA_Setup := 4;
		END_IF
		
	4:	//Homing stoppen
		fbAxisControl(Home := FALSE, Axis:= pAxisRef^);
		IF pAxisRef^.AxisState <> tenLM_AxisState.Homing_LM THEN
			nStateA_Setup := 5;
		END_IF
		
	5:	//HomingSpeed auf "0.02" setzen
		fbLMcfParaAccess(Execute:= TRUE , Mode:= 3, UPIDIn:=16#13C8 , Axis:= pAxisRef^, ValueIn := 20000);
		IF NOT fbLMcfParaAccess.Busy THEN
			IF fbLMcfParaAccess.Error THEN
				nErrorId := fbLMcfParaAccess.ErrorID;
				nStateA_Setup := 99;
			ELSE
				nStateA_Setup := 6;	
			END_IF
			fbLMcfParaAccess(Execute:= FALSE, Axis:= pAxisRef^);
		END_IF
		
	6:	//Achse ausschalten
		fbAxisControl(SwitchOn := FALSE, Axis:= pAxisRef^);
		IF NOT fbAxisControl.OperationEnabled THEN
			nStateA_Setup := 10; //Weiterschalten zu "11" verfolgt durch fb_OM_Maintenance
			bSetupWaitForResp := TRUE; //Wartet auf Antwort vom User
			bContinueSetup := FALSE;
		END_IF
		
	10: //Auf Antwort vom User warten, dass teaching beendet 
		IF bContinueSetup THEN
			nStateA_Setup := 11;
		ELSIF bStop THEN
			nStateA_Setup := 70;
		END_IF
		
	11:	//Referenzposition berechnen
		IF eXYOrientation = E_XYOrientation.X THEN
			rRefPosMaster := rWorkplateLength - P_rActPos - rSetupPosDist - rNullPosDist;
		ELSE
			rRefPosMaster := (-P_rActPos) + rSetupPosDist - rNullPosDist;
		END_IF
		nStateA_Setup := 80;
	
	70:	//Abbrechen
		fbLMcfParaAccess(Execute:= FALSE, Axis:= pAxisRef^);
		fbAxisControl(SwitchOn := FALSE, Home := FALSE, Axis:= pAxisRef^);
		nStateA_Setup := 80;
	
END_CASE
END_ACTION

METHOD M_Capture : ERRORID
VAR_INPUT
END_VAR
nCapturedCounterOld := nCapturedCounter;
bCapture := TRUE;
bCaptureOk := FALSE;
bCaptureStopped := FALSE;
A_Capture();
END_METHOD

ACTION A_Reset:
timeout();

CASE nStateA_Reset OF
	0:	
		IF timeout.Q THEN
			timeout(IN:= FALSE);
			fbLMcfParaAccess(Execute:= FALSE, Axis:= pAxisRef^);
			fbAxisControl.ErrorAcknowledge := FALSE;
			nStateA_Reset := 1;
			RETURN;
		END_IF

		//Achse im Fehlerzustand? -> Versuchen, durch "ErrorAcknowledge" zurückzusetzen
		//Fall nicht erfolgreich, dann die Achse resetten (nStateA_Reset = 1)
		IF fbAxisControl.Error THEN
			timeout(IN:= TRUE, PT:= T#2S);
			fbAxisControl(ErrorAcknowledge := TRUE, SwitchOn := FALSE, JogPlus:= FALSE, JogMinus:= FALSE, Home:= FALSE, Axis:= pAxisRef^);
		ELSE
			timeout(IN:= FALSE);
			fbAxisControl.ErrorAcknowledge := FALSE;
			nStateA_Reset := 3;
		END_IF
		
	1:	//Achse resetten
		fbCoeWrite(sNetId:= stAdsAddress.sNetId, nSlaveAddr:= stAdsAddress.nPort, nIndex:= 16#2000, nSubIndex:= 16#0B,
				pSrcBuf:= ADR(nCoeData), cbBufLen:= 0, tTimeout := T#10S, bExecute:= TRUE);
		IF NOT fbCoeWrite.bBusy THEN
			IF fbCoeWrite.bError THEN
				nStateA_Reset := 99;
			ELSE
				timeout(IN:= TRUE, PT:= T#15S); //Achse sollte sich spätestens nach 15sec. wieder melden
				nStateA_Reset := 2;
			END_IF
			fbCoeWrite(bExecute:= FALSE);
		END_IF
		
	2:	//Fehler zurückgesetzt?
		IF timeout.Q THEN
			timeout(IN:= FALSE);
			nStateA_Reset := 99;
		END_IF
		
		IF NOT fbAxisControl.Error THEN
			timeout(IN:= FALSE);
			nStateA_Reset := 3;
		END_IF

	3:	//Achse freigeben nur wenn vorher PowerOn war
		timeout(IN:= TRUE, PT:= T#3S);
		fbAxisControl(SwitchOn := TRUE,JogPlus:= FALSE, JogMinus:= FALSE, Axis:= pAxisRef^);
		IF fbAxisControl.OperationEnabled THEN
			timeout(IN:= FALSE);
			IF fbAxisControl.Error THEN
				nStateA_Reset := 99;
			ELSE
				nStateA_Reset := 80;
				bError := FALSE;
			END_IF
		END_IF
END_CASE
END_ACTION

ACTION A_Init:
CASE nStateA_Init OF
	0: //Achse einschalten, falls noch nicht an
		M_PowerOn();
		nStateA_Init := 1;

	1:	//PowerOn OK?
		IF bError THEN
			nStateA_Init := 99;
			RETURN;
		END_IF
		IF NOT bPowerOn THEN
			nStateA_Init := 2;
		END_IF

	2:	//Home-Position in Antrieb schreiben (RAM)
		IF eXYOrientation = E_XYOrientation.X THEN
			fbLMcfParaAccess.ValueIn := REAL_TO_DINT(rHomePos * -10.0);
		ELSE
			fbLMcfParaAccess.ValueIn := REAL_TO_DINT(rHomePos * 10.0);	
		END_IF
	
		fbLMcfParaAccess(Execute:= TRUE , Mode:= 3, UPIDIn:=16#13C7 , Axis:= pAxisRef^);
		IF NOT fbLMcfParaAccess.Busy THEN
			IF fbLMcfParaAccess.Error THEN
				nErrorId := fbLMcfParaAccess.ErrorID;
				nStateA_Init := 99;
			ELSE
				nStateA_Init := 3;
			END_IF
			fbLMcfParaAccess(Execute:= FALSE, Axis:= pAxisRef^);
		END_IF
		
	3:	//Slider-Home-Position in Antrieb schreiben (RAM)
		IF eXYOrientation = E_XYOrientation.X THEN
			fbLMcfParaAccess.ValueIn := REAL_TO_DINT(rHomePos * 10.0 + 378000.0);
		ELSE
			fbLMcfParaAccess.ValueIn := REAL_TO_DINT(rHomePos * 10.0 + 180000.0);
		END_IF
	
		fbLMcfParaAccess(Execute:= TRUE , Mode:= 3, UPIDIn:=16#13CA , Axis:= pAxisRef^);
		IF NOT fbLMcfParaAccess.Busy THEN
			IF fbLMcfParaAccess.Error THEN
				nErrorId := fbLMcfParaAccess.ErrorID;
				nStateA_Init := 99;
			ELSE
				nStateA_Init := 4;
			END_IF
			fbLMcfParaAccess(Execute:= FALSE, Axis:= pAxisRef^);
		END_IF
		
	4:	//Homing notwendig?
		IF NOT fbAxisControl.Homed OR bReInit THEN
			IF bInvertInitDir THEN
				fbLMcfParaAccess.ValueIn := 16#A;
			ELSE
				fbLMcfParaAccess.ValueIn := 16#B;
			END_IF
			nStateA_Init := 5;
		ELSE
			nStateA_Init := 80;
		END_IF
		
	5:	//Homing-Richtung
		fbLMcfParaAccess(Execute:= TRUE , Mode:= 3, UPIDIn:=16#13C4 , Axis:= pAxisRef^);
		IF NOT fbLMcfParaAccess.Busy THEN
			IF fbLMcfParaAccess.Error THEN
				nErrorId := fbLMcfParaAccess.ErrorID;
				nStateA_Init := 99;
			ELSE
				nStateA_Init := 6;
			END_IF
			fbLMcfParaAccess(Execute:= FALSE, Axis:= pAxisRef^);
		END_IF
		
	6:	//Homing
		IF bStop THEN
			fbAxisControl(Home := FALSE, Axis:= pAxisRef^);
			nStateA_Init := 70;
			RETURN;
		END_IF
		tmrHoming(IN:= TRUE,PT:= T#100S);
		fbAxisControl(Home := TRUE, Axis:= pAxisRef^);
		IF fbAxisControl.Homed THEN
			tmrHoming(IN:= FALSE);
			fbAxisControl(Home := FALSE, Axis:= pAxisRef^);
			nStateA_Init := 80;
		END_IF
		
		IF fbAxisControl.Error THEN
			nErrorId := fbAxisControl.ErrorCode;
			nStateA_Init := 99;
		END_IF
		
	70:	//Abbrechen
		fbLMcfParaAccess(Execute:= FALSE, Axis:= pAxisRef^);
		fbAxisControl(SwitchOn := FALSE, Home := FALSE, Axis:= pAxisRef^);
		tmrHoming(IN:= FALSE);
		nStateA_Init := 80;

	99:	//Error
		bBusy := FALSE;
		bError := TRUE;
		tmrHoming(IN:= FALSE);
END_CASE
END_ACTION

PROPERTY P_tHomingTime : TIME
GET
P_tHomingTime := tmrHoming.ET;
END_GET
END_PROPERTY

METHOD M_MoveRel : ERRORID
VAR_INPUT
	rDistance		: REAL;
	rSpeed			: REAL;
	rAcceleration 	: REAL;
	rDeceleration 	: REAL;
END_VAR
IF bBusy THEN
	M_MoveRel := E_ErrorIdCmd.ERRORID_AxisStillBusy;
ELSE
	IF rSpeed = 0 THEN
		RETURN;
	END_IF
	
	IF eXYOrientation = E_XYOrientation.X THEN //X - Achse hat negativen Hub
		fbLMmtMoveRel.Distance := rDistance / -1000.0;
	ELSE
		fbLMmtMoveRel.Distance := rDistance / 1000.0;	
	END_IF
	
	fbLMmtMoveRel.Velocity := rSpeed / 1000000.0;
	IF rAcceleration > 0.0 THEN
		fbLMmtMoveRel.Acceleration := rAcceleration / 1000000.0;
	ELSE
		fbLMmtMoveRel.Acceleration := 1.0;
	END_IF
	IF rDeceleration > 0.0 THEN
		fbLMmtMoveRel.Deceleration := rDeceleration / 1000000.0;
	ELSE
		fbLMmtMoveRel.Deceleration := 1.0;
	END_IF
	bMoveRel := TRUE;
	A_MoveRel();
END_IF
END_METHOD

ACTION A_MoveAbs:
IF fbLMmtMoveAbs.Error THEN
	nErrorId := UDINT_TO_UINT(fbLMmtMoveAbs.ErrorId);
	fbLMmtMoveAbs(Axis:= pAxisRef^, Execute:= FALSE);
	nStateMoveAbs := 99;
END_IF

CASE nStateMoveAbs OF
	0:
		IF bStop THEN
			nStateMoveAbs := 80;
		ELSE
			bBusy := TRUE;
			fbLMmtMoveAbs(Axis:= pAxisRef^, Execute:= TRUE);
			nStateMoveAbs := 1;
		END_IF
	
	1:	//Warten bis Move fertig
		IF bStop THEN
			fbLMmtStop(Execute:= TRUE, Axis:= pAxisRef^, Deceleration:= 1.0);
			fbLMmtMoveAbs(Axis:= pAxisRef^, Execute:= FALSE);
			nStateMoveAbs := 2;
		ELSE
			fbLMmtMoveAbs(Axis:= pAxisRef^);
			IF NOT fbLMmtMoveAbs.Busy THEN
				fbLMmtMoveAbs(Axis:= pAxisRef^, Execute:= FALSE);
				nStateMoveAbs := 80;
			END_IF			
		END_IF
	2:	//Warten bis Stop fertig
		IF fbLMmtStop.Error THEN
			bError := TRUE;
			nErrorId := fbLMmtStop.ErrorID;
			nStateMoveAbs := 99;
			bStop := FALSE;
		END_IF
		
		IF NOT fbLMmtStop.Busy THEN
			fbLMmtStop(Execute:= FALSE, Axis:= pAxisRef^);
			nStateMoveAbs := 80;
			bStop := FALSE;
		END_IF
END_CASE
END_ACTION

ACTION A_Jog:
IF fbLMmtMoveRel.Error THEN
	nErrorId := UDINT_TO_UINT(fbLMmtMoveRel.ErrorId);
	fbLMmtMoveRel(Axis:= pAxisRef^, Execute:= FALSE);
	nStateA_Jog := 99;
	bError := TRUE;
	bBusy := FALSE;
	RETURN;
END_IF

IF fbLMmtMoveAbs.Error THEN
	nErrorId := UDINT_TO_UINT(fbLMmtMoveAbs.ErrorId);
	fbLMmtMoveAbs(Axis:= pAxisRef^, Execute:= FALSE);
	nStateA_Jog := 99;
	bError := TRUE;
	bBusy := FALSE;
	RETURN;
END_IF

//Kontinuierliches Jogging mittels MoveAbs in Richtung Minimum bzw Maximum
//Inkrementelles Jogging mittels MoveRel (mit vorheriger Abfrage der Grenzen) 
CASE nStateA_Jog OF
	0:
		bBusy := TRUE;
		IF bJogInching THEN
			fbLMmtMoveRel(Axis:= pAxisRef^, Execute:= TRUE);
			nStateA_Jog := 1;
		ELSE
			fbLMmtMoveAbs(Axis:= pAxisRef^, Execute:= TRUE);
			nStateA_Jog := 2;
		END_IF
		
	2:	//Timer abfragen
		tmrJog(IN:= TRUE, PT:= T#500MS);
		IF tmrJog.Q THEN
			fbLMmtStop(Axis:= pAxisRef^, Execute:= TRUE, Deceleration:= 2.0);
			bError := TRUE;
		END_IF
		
	70:	//Stop
		fbLMmtStop(Axis:= pAxisRef^, Execute:= TRUE, Deceleration:= 2.0);
		
END_CASE

IF bJogInching THEN
	fbLMmtMoveRel(Axis:= pAxisRef^);
	IF NOT fbLMmtMoveRel.Busy THEN
		fbLMmtMoveRel(Axis:= pAxisRef^, Execute:= FALSE);
		
		//In Abhängigkeit von Ursache Stop in fertig oder wieder zu State"0"
		IF nStateA_Jog = 70 THEN
			IF NOT (bJogForward OR bJogBackward) THEN //geplanter Stop
				nStateA_Jog := 80;	
			ELSE //Stop durch Richtungsumkehr oder Umkehr des Modes
				nStateA_Jog := 0;
			END_IF
		ELSE
			nStateA_Jog := 80;
		END_IF
	END_IF
ELSE
	fbLMmtMoveAbs(Axis:= pAxisRef^);
	IF NOT fbLMmtMoveAbs.Busy THEN
		fbLMmtMoveAbs(Axis:= pAxisRef^, Execute:= FALSE);
		tmrJog(IN:= FALSE);
		nStateA_Jog := 80;
	END_IF	
END_IF
END_ACTION

METHOD M_MoveAbs : ERRORID
VAR_INPUT
	rPosition 		: REAL;
	rSpeed			: REAL;
	rAcceleration 	: REAL;
	rDeceleration 	: REAL;
END_VAR
IF bBusy THEN
	M_MoveAbs := E_ErrorIdCmd.ERRORID_AxisStillBusy;
ELSE
	IF rSpeed = 0 THEN
		RETURN;
	END_IF
	
	IF rPosition < P_rMinPos OR rPosition > P_rMaxPos THEN
		M_MoveAbs := E_ErrorIdCmd.ERRORID_TargetPosOutOfRangeX;
		RETURN;		
	END_IF
	
	IF eXYOrientation = E_XYOrientation.X THEN //X - Achse hat negativen Hub
		fbLMmtMoveAbs.Position := rPosition / -1000.0;
	ELSE
		fbLMmtMoveAbs.Position := rPosition / 1000.0;	
	END_IF

	fbLMmtMoveAbs.Velocity := rSpeed / 1000000.0;
	IF rAcceleration > 0.0 THEN
		fbLMmtMoveAbs.Acceleration := rAcceleration / 1000000.0;
	ELSE
		fbLMmtMoveAbs.Acceleration := 0.25;
	END_IF
	IF rDeceleration > 0.0 THEN
		fbLMmtMoveAbs.Deceleration := rDeceleration / 1000000.0;
	ELSE
		fbLMmtMoveAbs.Deceleration := 0.25;
	END_IF
	bMoveAbs := TRUE;
	A_MoveAbs();
END_IF
END_METHOD

METHOD M_PowerOff : ERRORID
VAR_INPUT
END_VAR
fbAxisControl(SwitchOn := FALSE,JogPlus:= FALSE, JogMinus:= FALSE, Axis:= pAxisRef^);
END_METHOD

ACTION A_StopCapture:
CASE nStateA_StopCapture OF
	0:	IF bCapture AND nStateA_Capture < 70 THEN
			nStateA_Capture := 70;
			nStateA_StopCapture := 1;
		ELSE
			nStateA_StopCapture := 80;
		END_IF
		
	1:	IF NOT bCapture THEN
			bCaptureStopped := TRUE;
			nStateA_StopCapture := 80;
		END_IF
END_CASE
END_ACTION

END_FUNCTION_BLOCK

// ---- Hardware/RS232/FB_SerialComPort_PC.TcPOU
FUNCTION_BLOCK FB_SerialComPort_PC EXTENDS FB_SerialComPort_Base
VAR_INPUT
END_VAR
VAR_OUTPUT
END_VAR
VAR
	InData	AT %I* 			: Tc2_SerialCom.PcComInData;
	OutData	AT %Q* 			: Tc2_SerialCom.PcComOutData;
	fbSerialLineControl 	: Tc2_SerialCom.SerialLineControl;
	nErrorIDSerialCom		: Tc2_SerialCom.ComError_t;
	nState					: USINT;	
END_VAR

SUPER^();
//wird direkt mit einem Hardware-Com-Port gemappt
IF nState = 0 THEN
	fbSerialLineControl(Mode:= Tc2_SerialCom.SERIALLINEMODE_DEFAULT,
					pComIn:= ADR(InData), 
					pComOut:= ADR(OutData), 
					SizeComIn:= DINT_TO_INT(SIZEOF(InData)), 
					ErrorID=> nErrorIDSerialCom, 
					TxBuffer:= TxBufferSerialCom, 
					RxBuffer:= RxBufferSerialCom );
	IF fbSerialLineControl.Error THEN
		nState := 99;
	END_IF				
END_IF

END_FUNCTION_BLOCK

// ---- Hardware/RS232/FB_SerialComPort_USB.TcPOU
FUNCTION_BLOCK FB_SerialComPort_USB EXTENDS FB_SerialComPort_Base
VAR_INPUT
END_VAR
VAR_OUTPUT
END_VAR
VAR
	nState : USINT;
	fbSerialLineControlADS 	: SerialLineControlADS;
	stComSerialConfig 		: ComSerialConfig := (ComPort:= 3);
	timer					: TON;
	nAttemps				: USINT;
END_VAR

SUPER^();
CASE nState OF
	0:	//Search virtual ComPort
		timer(IN:= TRUE, PT:= T#2S);
		IF timer.Q THEN
			fbSerialLineControlADS(Connect:= TRUE, SerialCfg:= stComSerialConfig, TxBuffer:= TxBufferSerialCom, RxBuffer:= RxBufferSerialCom);
			IF fbSerialLineControlADS.Error THEN
				IF fbSerialLineControlADS.ErrorID = 6 THEN	//Der SerialAdsServer ist noch nicht gestartet
					RETURN;
				END_IF
				IF fbSerialLineControlADS.ErrorID = 36915 THEN //Port schon connected
					RETURN;
				END_IF
				IF stComSerialConfig.ComPort = 6 THEN
					nAttemps := nAttemps + 1;
					stComSerialConfig.ComPort := 2; //Dadurch wird wieder bei 3 begonnen
					fbSerialLineControlADS(Connect:= FALSE, SerialCfg:= stComSerialConfig, TxBuffer:= TxBufferSerialCom, RxBuffer:= RxBufferSerialCom);
				END_IF
				stComSerialConfig.ComPort := stComSerialConfig.ComPort + 1;
			ELSE
				IF fbSerialLineControlADS.PortOpened THEN
					nState := 1;
				END_IF
			END_IF
		END_IF
	
	1: //Running
		fbSerialLineControlADS(Connect:= TRUE, SerialCfg:= stComSerialConfig, TxBuffer:= TxBufferSerialCom, RxBuffer:= RxBufferSerialCom);
		bIsWorking := TRUE;
		IF fbSerialLineControlADS.Error THEN
			fbSerialLineControlADS(Connect:= FALSE, SerialCfg:= stComSerialConfig, TxBuffer:= TxBufferSerialCom, RxBuffer:= RxBufferSerialCom);
		END_IF	
END_CASE

END_FUNCTION_BLOCK

// ---- Hardware/RS232/FB_SerialComPort_EL60xx.TcPOU
FUNCTION_BLOCK FB_SerialComPort_EL60xx EXTENDS FB_SerialComPort_Base
VAR_INPUT
END_VAR
VAR_OUTPUT
END_VAR
VAR
	InData	AT %I*			: EL6inData22B;
	OutData	AT %Q*			: EL6outData22B;
	fbSerialLineControl 	: Tc2_SerialCom.SerialLineControl;
	nErrorIDSerialCom		: Tc2_SerialCom.ComError_t;
	nState					: USINT;
END_VAR

SUPER^();
//wird direkt mit einem Hardware-Com-Port gemappt
IF nState = 0 THEN
	fbSerialLineControl(Mode:= Tc2_SerialCom.SERIALLINEMODE_EL6_22B,
					pComIn:= ADR(InData), 
					pComOut:= ADR(OutData), 
					SizeComIn:= DINT_TO_INT(SIZEOF(InData)), 
					ErrorID=> nErrorIDSerialCom, 
					TxBuffer:= TxBufferSerialCom, 
					RxBuffer:= RxBufferSerialCom);
	IF fbSerialLineControl.Error THEN
		nState := 99;
	END_IF				
END_IF

END_FUNCTION_BLOCK

// ---- Actions/FB_ComplexAction.TcPOU
FUNCTION_BLOCK FB_ComplexAction

VAR_OUTPUT
	bBusy				: BOOL;
	bError				: BOOL;
	nErrorId			: ERRORID;
	eCurrentState		: E_MachineState := E_MachineState.MACHINESTATE_Idle;
END_VAR

VAR
	//Variablen allgemeine Statemachine
	stError				: ST_Error;
	bInternCanceled		: BOOL;
	bPauseRequestIntern	: BOOL;	//Weiterleitung an ActionDispacher dann an Sequence
								//ermöglicht einer Action, welche aus einer Sequence aufgerufen wurde, diese in Pause zu versetzen
	bLastActionResult	: BOOL;
	nLastActionResult	: DINT;	//wird nur von ausgewählten ComplexActions zurückgegeben
	
	
	nActionState		: USINT;
	nActionStateNext	: USINT;
	
	bStop				: BOOL;
	
	eCurrentAction		: E_Action;
	
	//*****************************************ObjectPointer*****************************************************
	pMzTool					: POINTER TO FB_MzTool;
	pZLevelSensor			: POINTER TO FB_ZLevelSensor;
	pStampSupport			: POINTER TO FB_StampSupport;
	pPiezoPip				: POINTER TO FB_PiezoPip;
	pPassivePip				: POINTER TO FB_PassivPip;
	pLuer					: POINTER TO FB_Luer;
	pLuer2					: POINTER TO FB_Luer;
	pTriplePip				: POINTER TO FB_TriplePip;
	pDiluter1				: POINTER TO FB_Diluter;
	pDiluter2				: POINTER TO FB_Diluter;
	pTwinPiezoHolder		: POINTER TO FB_TwinPiezoHolder;
	pSolenoidPip			: POINTER TO FB_SolenoidPip;
	pVacuumHandler			: POINTER TO FB_VacuumHandler;
	ppHElectrode			: POINTER TO FB_pHElectrode;
	pHybridDispenser		: POINTER TO FB_HybridDispenser;
	pMultiCartHolder		: POINTER TO FB_MultiCartHolder;
	pExtruder				: POINTER TO FB_Extruder;
	pTwinExtruder			: POINTER TO FB_TwinExtruder;
	pGripper				: POINTER TO FB_Gripper;
	
	pTarget					: POINTER TO FB_TargetBase;
	pArray					: POINTER TO FB_Array;
	pInkStation				: POINTER TO FB_InkStation;
	pTipCalibrator			: POINTER TO FB_TipCalibrator;
	pTipCleaner				: POINTER TO FB_TipCleaner;
	pTipCleanerGen2			: POINTER TO FB_TipCleanerGen2;
	pStampMagazine			: POINTER TO FB_StampMagazine;
	pWashStation			: POINTER TO FB_WashStation;
	pMtp					: POINTER TO FB_Mtp;
	pDryPad					: POINTER TO FB_DryPad;
	pStroboscope			: POINTER TO FB_Stroboscope;
	pRack					: POINTER TO FB_Rack;
	pNeedleRack				: POINTER TO FB_NeedleRack;
	pFlipTubeRack			: POINTER TO FB_FlipTubeRack;
	pReactor				: POINTER TO FB_Reactor;
	pPowderStation			: POINTER TO FB_PowderStation;
	pHighVoltTray			: POINTER TO FB_HighVoltTray;
	ppHElectrCapRack		: POINTER TO FB_pHElectrodeCapRack;
	pSlide					: POINTER TO FB_Slide;
	pCartDispenser			: POINTER TO FB_CartDispenser;
	pTrayTransporter		: POINTER TO FB_TrayTransporter;
	
	pPiece					: POINTER TO FB_PieceBase;
	pSlot					: POINTER TO FB_Slot;
	pPieceSlot				: POINTER TO FB_PieceSlot;
	pNeedle					: POINTER TO FB_Needle;
	pTip					: POINTER TO FB_Tip;
	pFlipTube				: POINTER TO FB_FlipTube;
	pVial					: POINTER TO FB_Vial;
	pNozzle					: POINTER TO FB_Nozzle;
	
	iTargetZSensor			: I_TargetZSensor;
	iUsingDryPad			: I_UsingDryPad;
	iDispenser				: I_Dispenser;
	
	pSequence				: POINTER TO FB_Sequence;
	
	//****************************************Aktionvariablen****************************************************
	i						: UINT;
	bFlag					: BOOL; //Flag zur allgemeinen Verwendung
	bSingleStep				: BOOL;
	bSingleStepContinue		: BOOL;
	nSingleStepNextState	: USINT;
	
	eAction					: E_Action;
	stActionData			: ST_ActionData;
	stActionData2			: ST_ActionData;
	nCol					: UINT;
	nRow					: UINT;
	nSpecPointSlotNr		: UINT;
	stPoint1 				: ST_3DPoint;
	stPoint2 				: ST_3DPoint;
	stDimension				: ST_3DDimension;
	nZOffset1				: DINT;
	nZOffset2				: DINT;
	nZOffset3				: DINT;
	nDistance1				: DINT;
	nSpeed1					: DINT;
	rSumDockOffset			: REAL;	//Summe von DockOffset Tool und Piece
	
